KUKA KRL program: MyProgram_102().src

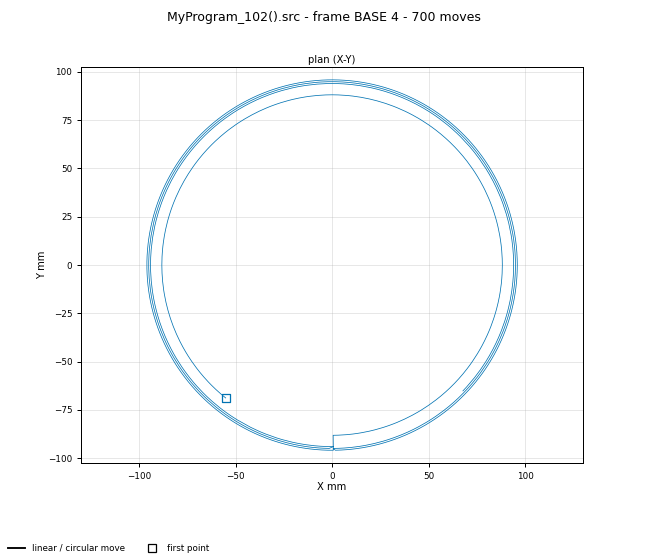
[picture p0: tool path of MyProgram_102().src in frame BASE 4, 700 of 700 moves have a stored position in this frame; points joined in program order, loops and branches not executed]
&ACCESS RVP
&REL 1
&PARAM TEMPLATE = C:\KRC\Roboter\Template\vorgabe
&PARAM EDITMASK = *
DEF MyProgram_102()
; ---- Setting reference (Base) ----
$BASE = BASE_DATA[4]

; --------------------------
; ---- Setting tool (TCP) ----
$TOOL = TOOL_DATA[3]
; --------------------------

$VEL.CP = VEL_APROX_PRINT
Startdeposition()
$VEL.CP = VEL_PRINT
LIN {X -55.0908,Y -68.8006,Z 92,A -133.8998,B 24.9282,C -1.9576,E1 24.8989,E2 -141.0227} C_DIS
LIN {X -57.6205,Y -66.6959,Z 92,A -136.0232,B 24.9278,C -1.9621,E1 24.8943,E2 -138.9019} C_DIS
LIN {X -60.1121,Y -64.4587,Z 92,A -138.1865,B 24.9275,C -1.9669,E1 24.8899,E2 -136.7412} C_DIS
LIN {X -62.4,Y -62.2469,Z 92,A -140.2884,B 24.9272,C -1.9702,E1 24.8857,E2 -134.6384} C_DIS
LIN {X -64.1532,Y -60.4369,Z 92,A -141.8968,B 24.9269,C -1.9746,E1 24.8826,E2 -133.0336} C_DIS
LIN {X -66.3939,Y -57.9664,Z 92,A -144.0684,B 24.9265,C -1.9794,E1 24.8786,E2 -130.8637} C_DIS
LIN {X -68.514,Y -55.4444,Z 92,A -146.1669,B 24.9261,C -1.9856,E1 24.8748,E2 -128.7703} C_DIS
LIN {X -70.1385,Y -53.3772,Z 92,A -147.8949,B 24.9258,C -1.9891,E1 24.8719,E2 -127.0425} C_DIS
LIN {X -71.5084,Y -51.5264,Z 92,A -149.3014,B 24.9253,C -1.9955,E1 24.8696,E2 -125.6443} C_DIS
LIN {X -72.6787,Y -49.8632,Z 92,A -150.8425,B 24.9256,C -1.9924,E1 24.8671,E2 -124.0882} C_DIS
LIN {X -74.4672,Y -47.1505,Z 92,A -152.7543,B 24.9247,C -2.0036,E1 24.8642,E2 -122.1936} C_DIS
LIN {X -75.8238,Y -44.9334,Z 92,A -154.6554,B 24.9249,C -2.002,E1 24.8615,E2 -120.2787} C_DIS
LIN {X -77.2426,Y -42.4507,Z 92,A -156.5523,B 24.9246,C -2.0058,E1 24.8589,E2 -118.3811} C_DIS
LIN {X -78.7875,Y -39.5087,Z 92,A -158.4218,B 24.9235,C -2.0202,E1 24.8565,E2 -116.5359} C_DIS
LIN {X -79.732,Y -37.5663,Z 92,A -159.8342,B 24.9232,C -2.0238,E1 24.8548,E2 -115.1246} C_DIS
LIN {X -80.5782,Y -35.7169,Z 92,A -161.3104,B 24.9232,C -2.0231,E1 24.8531,E2 -113.6385} C_DIS
LIN {X -81.475,Y -33.6191,Z 92,A -162.7506,B 24.9228,C -2.0286,E1 24.8516,E2 -112.2034} C_DIS
LIN {X -82.2377,Y -31.7093,Z 92,A -164.0784,B 24.9225,C -2.0327,E1 24.8502,E2 -110.878} C_DIS
LIN {X -83.0309,Y -29.5683,Z 92,A -165.5727,B 24.9222,C -2.0368,E1 24.8488,E2 -109.385} C_DIS
LIN {X -83.691,Y -27.6469,Z 92,A -166.9707,B 24.9221,C -2.0385,E1 24.8476,E2 -107.983} C_DIS
LIN {X -84.3756,Y -25.4792,Z 92,A -168.4079,B 24.9216,C -2.0441,E1 24.8464,E2 -106.5509} C_DIS
LIN {X -84.9491,Y -23.4984,Z 92,A -169.9139,B 24.9217,C -2.0434,E1 24.8452,E2 -105.0346} C_DIS
LIN {X -85.5268,Y -21.2978,Z 92,A -171.2261,B 24.921,C -2.0527,E1 24.8443,E2 -103.7368} C_DIS
LIN {X -85.9938,Y -19.3285,Z 92,A -172.5544,B 24.9207,C -2.0563,E1 24.8435,E2 -102.4095} C_DIS
LIN {X -86.4685,Y -17.077,Z 92,A -174.0675,B 24.9204,C -2.0605,E1 24.8427,E2 -100.8973} C_DIS
LIN {X -86.8426,Y -15.0633,Z 92,A -175.4002,B 24.9201,C -2.0646,E1 24.842,E2 -99.5665} C_DIS
LIN {X -87.1856,Y -12.931,Z 92,A -176.8138,B 24.9197,C -2.0687,E1 24.8414,E2 -98.1543} C_DIS
LIN {X -87.4909,Y -10.6657,Z 92,A -178.3106,B 24.9194,C -2.0731,E1 24.8409,E2 -96.659} C_DIS
LIN {X -87.726,Y -8.5188,Z 92,A -179.6515,B 24.9189,C -2.0793,E1 24.8405,E2 -95.3249} C_DIS
LIN {X -87.9265,Y -6.0991,Z 92,A 178.8138,B 24.9184,C -2.0855,E1 24.8401,E2 -93.7959} C_DIS
LIN {X -88.0388,Y -4.1929,Z 92,A 177.5128,B 24.9183,C -2.0878,E1 24.8399,E2 -92.4925} C_DIS
LIN {X -88.1151,Y -2.0351,Z 92,A 176.0233,B 24.9181,C -2.0898,E1 24.8399,E2 -90.9988} C_DIS
LIN {X -88.139,Y -0.0018,Z 92,A 174.7078,B 24.9178,C -2.0942,E1 24.8398,E2 -89.6858} C_DIS
LIN {X -88.1091,Y 2.2827,Z 92,A 173.2673,B 24.9173,C -2.1002,E1 24.8398,E2 -88.2511} C_DIS
LIN {X -88.0328,Y 4.3304,Z 92,A 171.7854,B 24.9173,C -2.1002,E1 24.84,E2 -86.7603} C_DIS
LIN {X -87.8451,Y 7.1771,Z 92,A 169.9225,B 24.9168,C -2.106,E1 24.8404,E2 -84.8999} C_DIS
LIN {X -87.6023,Y 9.7143,Z 92,A 168.2489,B 24.9164,C -2.1108,E1 24.8409,E2 -83.2277} C_DIS
LIN {X -87.3205,Y 11.9815,Z 92,A 166.5136,B 24.9166,C -2.1085,E1 24.8415,E2 -81.4766} C_DIS
LIN {X -86.8138,Y 15.2235,Z 92,A 164.4771,B 24.9159,C -2.118,E1 24.8425,E2 -79.4507} C_DIS
LIN {X -86.1961,Y 18.4018,Z 92,A 162.6299,B 24.9148,C -2.132,E1 24.8435,E2 -77.6259} C_DIS
LIN {X -85.7502,Y 20.3818,Z 92,A 161.158,B 24.9148,C -2.1318,E1 24.8444,E2 -76.1451} C_DIS
LIN {X -85.1932,Y 22.595,Z 92,A 159.8078,B 24.9141,C -2.1403,E1 24.8453,E2 -74.8072} C_DIS
LIN {X -84.6148,Y 24.6728,Z 92,A 158.2368,B 24.9141,C -2.1399,E1 24.8466,E2 -73.226} C_DIS
LIN {X -83.6925,Y 27.6422,Z 92,A 156.2829,B 24.9135,C -2.1481,E1 24.8482,E2 -71.2805} C_DIS
LIN {X -82.9482,Y 29.7998,Z 92,A 154.7907,B 24.9131,C -2.1524,E1 24.8496,E2 -69.7902} C_DIS
LIN {X -82.0355,Y 32.2245,Z 92,A 152.9841,B 24.913,C -2.1541,E1 24.8514,E2 -67.9775} C_DIS
LIN {X -80.8405,Y 35.1151,Z 92,A 151.1415,B 24.912,C -2.1657,E1 24.8534,E2 -66.1523} C_DIS
LIN {X -79.6031,Y 37.8382,Z 92,A 149.1721,B 24.9116,C -2.1708,E1 24.8557,E2 -64.1843} C_DIS
LIN {X -78.7225,Y 39.6396,Z 92,A 147.6445,B 24.9118,C -2.1682,E1 24.8576,E2 -62.6423} C_DIS
LIN {X -77.6641,Y 41.6736,Z 92,A 146.2785,B 24.9112,C -2.1761,E1 24.8593,E2 -61.2879} C_DIS
LIN {X -76.6219,Y 43.5602,Z 92,A 144.9444,B 24.9107,C -2.1821,E1 24.8612,E2 -59.9611} C_DIS
LIN {X -75.5337,Y 45.4211,Z 92,A 143.5333,B 24.9104,C -2.1858,E1 24.8632,E2 -58.5516} C_DIS
LIN {X -74.4003,Y 47.2548,Z 92,A 141.9678,B 24.9104,C -2.1851,E1 24.8655,E2 -56.9763} C_DIS
LIN {X -73.1491,Y 49.1685,Z 92,A 140.635,B 24.9097,C -2.1936,E1 24.8675,E2 -55.6572} C_DIS
LIN {X -72.0234,Y 50.8046,Z 92,A 139.1962,B 24.9098,C -2.1929,E1 24.8698,E2 -54.2096} C_DIS
LIN {X -70.701,Y 52.6286,Z 92,A 137.6109,B 24.9098,C -2.1934,E1 24.8725,E2 -52.6178} C_DIS
LIN {X -68.8213,Y 55.065,Z 92,A 135.5536,B 24.9095,C -2.197,E1 24.876,E2 -50.5594} C_DIS
LIN {X -66.7411,Y 57.5688,Z 92,A 133.442,B 24.909,C -2.2026,E1 24.8798,E2 -48.4515} C_DIS
LIN {X -64.6768,Y 59.8775,Z 92,A 131.3966,B 24.9087,C -2.2067,E1 24.8837,E2 -46.4068} C_DIS
LIN {X -62.3288,Y 62.3189,Z 92,A 129.1613,B 24.9083,C -2.211,E1 24.888,E2 -44.1723} C_DIS
LIN {X -60.3328,Y 64.2511,Z 92,A 127.3713,B 24.9079,C -2.2157,E1 24.8917,E2 -42.3862} C_DIS
LIN {X -57.8348,Y 66.5088,Z 92,A 125.2447,B 24.9073,C -2.2225,E1 24.8961,E2 -40.2673} C_DIS
LIN {X -55.4085,Y 68.5431,Z 92,A 123.1721,B 24.907,C -2.2266,E1 24.9005,E2 -38.1966} C_DIS
LIN {X -53.2048,Y 70.2681,Z 92,A 121.5765,B 24.9061,C -2.237,E1 24.904,E2 -36.6199} C_DIS
LIN {X -51.4953,Y 71.5306,Z 92,A 120.1031,B 24.9061,C -2.2371,E1 24.9074,E2 -35.1416} C_DIS
LIN {X -49.8396,Y 72.6947,Z 92,A 118.7813,B 24.9059,C -2.2395,E1 24.9104,E2 -33.8211} C_DIS
LIN {X -48.05,Y 73.8899,Z 92,A 117.1497,B 24.9063,C -2.2354,E1 24.9142,E2 -32.1742} C_DIS
LIN {X -45.2023,Y 75.6648,Z 92,A 115.2604,B 24.9052,C -2.248,E1 24.9187,E2 -30.3092} C_DIS
LIN {X -43.4499,Y 76.6853,Z 92,A 113.8593,B 24.9052,C -2.2479,E1 24.9221,E2 -28.9035} C_DIS
LIN {X -41.4529,Y 77.7823,Z 92,A 112.3756,B 24.905,C -2.2503,E1 24.9257,E2 -27.4215} C_DIS
LIN {X -39.508,Y 78.7879,Z 92,A 111.0212,B 24.9046,C -2.2547,E1 24.9291,E2 -26.0738} C_DIS
LIN {X -37.5665,Y 79.7319,Z 92,A 109.6134,B 24.9045,C -2.2567,E1 24.9326,E2 -24.6673} C_DIS
LIN {X -35.7178,Y 80.5778,Z 92,A 108.0849,B 24.9048,C -2.2525,E1 24.9365,E2 -23.125} C_DIS
LIN {X -33.7201,Y 81.4339,Z 92,A 106.7186,B 24.9045,C -2.2559,E1 24.94,E2 -21.7637} C_DIS
LIN {X -31.6873,Y 82.2461,Z 92,A 105.3688,B 24.9042,C -2.26,E1 24.9435,E2 -20.4208} C_DIS
LIN {X -29.2147,Y 83.155,Z 92,A 103.5195,B 24.9043,C -2.2581,E1 24.9484,E2 -18.5632} C_DIS
LIN {X -26.4901,Y 84.0636,Z 92,A 101.8544,B 24.9036,C -2.2664,E1 24.9528,E2 -16.9148} C_DIS
LIN {X -24.4281,Y 84.6858,Z 92,A 100.4479,B 24.9036,C -2.2677,E1 24.9566,E2 -15.5091} C_DIS
LIN {X -22.4732,Y 85.2261,Z 92,A 98.9898,B 24.9038,C -2.2648,E1 24.9605,E2 -14.0418} C_DIS
LIN {X -20.2625,Y 85.778,Z 92,A 97.4007,B 24.9039,C -2.2629,E1 24.9648,E2 -12.4461} C_DIS
LIN {X -17.1934,Y 86.4461,Z 92,A 95.2808,B 24.9039,C -2.2622,E1 24.9706,E2 -10.3221} C_DIS
LIN {X -13.9877,Y 87.0222,Z 92,A 93.4019,B 24.9032,C -2.2711,E1 24.9758,E2 -8.4624} C_DIS
LIN {X -11.8524,Y 87.3387,Z 92,A 91.9278,B 24.9033,C -2.2698,E1 24.9799,E2 -6.984} C_DIS
LIN {X -9.5843,Y 87.6159,Z 92,A 90.5083,B 24.9031,C -2.2727,E1 24.9838,E2 -5.5705} C_DIS
LIN {X -7.561,Y 87.8144,Z 92,A 89.0193,B 24.9035,C -2.2681,E1 24.9879,E2 -4.0699} C_DIS
LIN {X -5.258,Y 87.9816,Z 92,A 87.6833,B 24.903,C -2.2739,E1 24.9916,E2 -2.7471} C_DIS
LIN {X -3.2295,Y 88.08,Z 92,A 86.1609,B 24.9035,C -2.268,E1 24.9959,E2 -1.2104} C_DIS
LIN {X 0.0063,Y 88.1393,Z 92,A 84.0319,B 24.9035,C -2.2677,E1 25.0019,E2 0.9194} C_DIS
LIN {X 3.2426,Y 88.0796,Z 92,A 82.1507,B 24.9029,C -2.2749,E1 25.0071,E2 2.783} C_DIS
LIN {X 5.712,Y 87.9527,Z 92,A 80.6353,B 24.9027,C -2.2778,E1 25.0113,E2 4.2909} C_DIS
LIN {X 7.6239,Y 87.8086,Z 92,A 79.1484,B 24.9033,C -2.2701,E1 25.0155,E2 5.7953} C_DIS
LIN {X 10.6692,Y 87.4905,Z 92,A 77.2297,B 24.9031,C -2.2721,E1 25.0208,E2 7.708} C_DIS
LIN {X 13.059,Y 87.1658,Z 92,A 75.741,B 24.903,C -2.2742,E1 25.0249,E2 9.1903} C_DIS
LIN {X 15.0667,Y 86.842,Z 92,A 74.4194,B 24.903,C -2.2738,E1 25.0285,E2 10.5117} C_DIS
LIN {X 17.3273,Y 86.4186,Z 92,A 72.811,B 24.9034,C -2.2695,E1 25.0329,E2 12.1282} C_DIS
LIN {X 19.4335,Y 85.9695,Z 92,A 71.5506,B 24.903,C -2.2733,E1 25.0363,E2 13.378} C_DIS
LIN {X 21.5838,Y 85.4548,Z 92,A 70.1059,B 24.9031,C -2.2722,E1 25.0403,E2 14.8231} C_DIS
LIN {X 23.5283,Y 84.9408,Z 92,A 68.7213,B 24.9034,C -2.2689,E1 25.044,E2 16.2135} C_DIS
LIN {X 25.5972,Y 84.3404,Z 92,A 67.3223,B 24.9035,C -2.2679,E1 25.0478,E2 17.6123} C_DIS
LIN {X 27.6515,Y 83.6895,Z 92,A 65.9918,B 24.9035,C -2.2691,E1 25.0513,E2 18.9376} C_DIS
LIN {X 29.8076,Y 82.9453,Z 92,A 64.4996,B 24.9035,C -2.2675,E1 25.0552,E2 20.4305} C_DIS
LIN {X 31.7317,Y 82.2291,Z 92,A 63.1111,B 24.9038,C -2.2644,E1 25.0588,E2 21.8233} C_DIS
LIN {X 33.7362,Y 81.4273,Z 92,A 61.7105,B 24.9039,C -2.2631,E1 25.0625,E2 23.2238} C_DIS
LIN {X 35.8356,Y 80.5247,Z 92,A 60.3722,B 24.9036,C -2.2663,E1 25.0659,E2 24.5513} C_DIS
LIN {X 37.7974,Y 79.6227,Z 92,A 58.9707,B 24.9038,C -2.2647,E1 25.0694,E2 25.953} C_DIS
LIN {X 39.6242,Y 78.7303,Z 92,A 57.5772,B 24.9041,C -2.2607,E1 25.0729,E2 27.3523} C_DIS
LIN {X 41.6636,Y 77.6695,Z 92,A 55.9506,B 24.9047,C -2.2544,E1 25.077,E2 28.9892} C_DIS
LIN {X 44.3912,Y 76.1443,Z 92,A 53.9967,B 24.9047,C -2.2541,E1 25.0817,E2 30.938} C_DIS
LIN {X 46.2391,Y 75.0365,Z 92,A 52.4841,B 24.9052,C -2.2482,E1 25.0853,E2 32.4596} C_DIS
LIN {X 48.1741,Y 73.8084,Z 92,A 51.1819,B 24.9048,C -2.2521,E1 25.0883,E2 33.7484} C_DIS
LIN {X 49.969,Y 72.6052,Z 92,A 49.7984,B 24.905,C -2.2506,E1 25.0915,E2 35.1309} C_DIS
LIN {X 51.792,Y 71.3158,Z 92,A 48.3444,B 24.9052,C -2.248,E1 25.0948,E2 36.586} C_DIS
LIN {X 53.8698,Y 69.7589,Z 92,A 46.5669,B 24.9057,C -2.242,E1 25.0988,E2 38.3711} C_DIS
LIN {X 56.3278,Y 67.7896,Z 92,A 44.4846,B 24.9061,C -2.237,E1 25.1033,E2 40.4574} C_DIS
LIN {X 58.7884,Y 65.6672,Z 92,A 42.4033,B 24.9064,C -2.2339,E1 25.1077,E2 42.5378} C_DIS
LIN {X 61.1617,Y 63.4625,Z 92,A 40.3127,B 24.9067,C -2.2301,E1 25.1119,E2 44.6288} C_DIS
LIN {X 63.584,Y 61.0357,Z 92,A 38.0714,B 24.9071,C -2.2249,E1 25.1163,E2 46.8728} C_DIS
LIN {X 65.6906,Y 58.7622,Z 92,A 36.0882,B 24.9074,C -2.2215,E1 25.1201,E2 48.8552} C_DIS
LIN {X 67.7931,Y 56.3236,Z 92,A 33.9988,B 24.9078,C -2.2168,E1 25.1238,E2 50.9463} C_DIS
LIN {X 69.8171,Y 53.7943,Z 92,A 31.9054,B 24.9082,C -2.2122,E1 25.1275,E2 53.0407} C_DIS
LIN {X 71.5065,Y 51.5289,Z 92,A 30.1759,B 24.9082,C -2.2114,E1 25.1303,E2 54.7639} C_DIS
LIN {X 72.6868,Y 49.8513,Z 92,A 28.8639,B 24.9085,C -2.2087,E1 25.1324,E2 56.0757} C_DIS
LIN {X 73.8818,Y 48.0627,Z 92,A 27.4051,B 24.909,C -2.2031,E1 25.1346,E2 57.5406} C_DIS
LIN {X 75.336,Y 45.7465,Z 92,A 25.6046,B 24.9094,C -2.1977,E1 25.1373,E2 59.3447} C_DIS
LIN {X 76.8415,Y 43.1704,Z 92,A 23.6162,B 24.91,C -2.1908,E1 25.1401,E2 61.3391} C_DIS
LIN {X 78.2963,Y 40.4734,Z 92,A 21.7949,B 24.91,C -2.1912,E1 25.1424,E2 63.1497} C_DIS
LIN {X 79.2093,Y 38.6577,Z 92,A 20.4139,B 24.9104,C -2.1855,E1 25.1442,E2 64.537} C_DIS
LIN {X 80.2289,Y 36.4919,Z 92,A 19.0306,B 24.9103,C -2.1871,E1 25.1458,E2 65.9089} C_DIS
LIN {X 81.0773,Y 34.5667,Z 92,A 17.6529,B 24.9106,C -2.1828,E1 25.1473,E2 67.2891} C_DIS
LIN {X 81.894,Y 32.5847,Z 92,A 16.2686,B 24.9109,C -2.1791,E1 25.1488,E2 68.6745} C_DIS
LIN {X 82.8407,Y 30.0945,Z 92,A 14.2939,B 24.912,C -2.1656,E1 25.1507,E2 70.6702} C_DIS
LIN {X 83.6873,Y 27.6579,Z 92,A 12.5817,B 24.9125,C -2.1594,E1 25.1522,E2 72.3875} C_DIS
LIN {X 84.6867,Y 24.4251,Z 92,A 10.6947,B 24.9122,C -2.1637,E1 25.1537,E2 74.2535} C_DIS
LIN {X 85.2283,Y 22.465,Z 92,A 9.2385,B 24.9129,C -2.1549,E1 25.1548,E2 75.7219} C_DIS
LIN {X 85.8933,Y 19.7634,Z 92,A 7.4194,B 24.9134,C -2.1491,E1 25.156,E2 77.5444} C_DIS
LIN {X 86.4709,Y 17.0642,Z 92,A 5.7273,B 24.9135,C -2.1471,E1 25.1569,E2 79.2314} C_DIS
LIN {X 86.8421,Y 15.0658,Z 92,A 4.4151,B 24.9138,C -2.1433,E1 25.1576,E2 80.5449} C_DIS
LIN {X 87.1851,Y 12.9345,Z 92,A 3.0201,B 24.9142,C -2.1391,E1 25.1582,E2 81.9414} C_DIS
LIN {X 87.5401,Y 10.2459,Z 92,A 1.1621,B 24.9149,C -2.1303,E1 25.1588,E2 83.8093} C_DIS
LIN {X 87.8161,Y 7.5401,Z 92,A -0.4838,B 24.9149,C -2.1289,E1 25.1593,E2 85.4486} C_DIS
LIN {X 87.9811,Y 5.2664,Z 92,A -1.9741,B 24.9154,C -2.1239,E1 25.1596,E2 86.9419} C_DIS
LIN {X 88.0797,Y 3.24,Z 92,A -3.4659,B 24.9162,C -2.1136,E1 25.1597,E2 88.4491} C_DIS
LIN {X 88.1389,Y 0.0069,Z 92,A -5.3507,B 24.9162,C -2.1145,E1 25.1597,E2 90.3205} C_DIS
LIN {X 88.1084,Y -2.3048,Z 92,A -6.7714,B 24.9162,C -2.1126,E1 25.1597,E2 91.7373} C_DIS
LIN {X 88.0326,Y -4.3342,Z 92,A -8.2242,B 24.917,C -2.1037,E1 25.1595,E2 93.2026} C_DIS
LIN {X 87.8575,Y -7.0222,Z 92,A -10.0056,B 24.9175,C -2.097,E1 25.1592,E2 94.9892} C_DIS
LIN {X 87.6028,Y -9.7095,Z 92,A -11.7033,B 24.9178,C -2.0934,E1 25.1587,E2 96.6854} C_DIS
LIN {X 87.29,Y -12.1961,Z 92,A -13.154,B 24.9178,C -2.0945,E1 25.1582,E2 98.125} C_DIS
LIN {X 86.9984,Y -14.1314,Z 92,A -14.4445,B 24.9181,C -2.0897,E1 25.1576,E2 99.4191} C_DIS
LIN {X 86.5651,Y -16.575,Z 92,A -16.2682,B 24.9191,C -2.0772,E1 25.1567,E2 101.2617} C_DIS
LIN {X 85.912,Y -19.6825,Z 92,A -18.3634,B 24.9197,C -2.0695,E1 25.1554,E2 103.3627} C_DIS
LIN {X 85.1708,Y -22.6778,Z 92,A -20.0757,B 24.9194,C -2.0735,E1 25.1543,E2 105.0557} C_DIS
LIN {X 84.5682,Y -24.8298,Z 92,A -21.7542,B 24.9203,C -2.061,E1 25.153,E2 106.7541} C_DIS
LIN {X 83.6823,Y -27.6728,Z 92,A -23.5261,B 24.9203,C -2.0607,E1 25.1515,E2 108.5167} C_DIS
LIN {X 82.9399,Y -29.8225,Z 92,A -24.9955,B 24.9207,C -2.0565,E1 25.1501,E2 109.9879} C_DIS
LIN {X 82.2338,Y -31.7197,Z 92,A -26.3809,B 24.9212,C -2.05,E1 25.1487,E2 111.381} C_DIS
LIN {X 81.4257,Y -33.7399,Z 92,A -27.7764,B 24.9215,C -2.0463,E1 25.1472,E2 112.7774} C_DIS
LIN {X 80.3531,Y -36.2164,Z 92,A -29.5599,B 24.922,C -2.04,E1 25.1452,E2 114.566} C_DIS
LIN {X 78.959,Y -39.1628,Z 92,A -31.6587,B 24.9224,C -2.0344,E1 25.1427,E2 116.6667} C_DIS
LIN {X 77.6798,Y -41.6448,Z 92,A -33.3604,B 24.9224,C -2.033,E1 25.1405,E2 118.3628} C_DIS
LIN {X 76.6385,Y -43.5313,Z 92,A -34.6938,B 24.9226,C -2.0313,E1 25.1387,E2 119.6933} C_DIS
LIN {X 75.271,Y -45.8533,Z 92,A -36.6436,B 24.9235,C -2.0194,E1 25.1358,E2 121.6612} C_DIS
LIN {X 73.8066,Y -48.1767,Z 92,A -38.2687,B 24.9235,C -2.0199,E1 25.1334,E2 123.2769} C_DIS
LIN {X 72.6762,Y -49.8669,Z 92,A -39.5825,B 24.9238,C -2.0165,E1 25.1313,E2 124.5923} C_DIS
LIN {X 71.3581,Y -51.7343,Z 92,A -41.0595,B 24.924,C -2.0127,E1 25.1289,E2 126.0709} C_DIS
LIN {X 69.7778,Y -53.8452,Z 92,A -42.8608,B 24.9246,C -2.0051,E1 25.1259,E2 127.8817} C_DIS
LIN {X 67.7817,Y -56.3373,Z 92,A -44.9696,B 24.9251,C -1.9985,E1 25.1222,E2 129.9963} C_DIS
LIN {X 65.666,Y -58.7897,Z 92,A -47.0296,B 24.9254,C -1.9947,E1 25.1184,E2 132.0561} C_DIS
LIN {X 63.4614,Y -61.1628,Z 92,A -49.1654,B 24.9259,C -1.9884,E1 25.1143,E2 134.1974} C_DIS
LIN {X 61.1128,Y -63.5097,Z 92,A -51.2854,B 24.9262,C -1.9845,E1 25.11,E2 136.3177} C_DIS
LIN {X 58.7852,Y -65.67,Z 92,A -53.3251,B 24.9265,C -1.9806,E1 25.1058,E2 138.3585} C_DIS
LIN {X 56.3325,Y -67.7856,Z 92,A -55.4211,B 24.9268,C -1.9762,E1 25.1014,E2 140.4568} C_DIS
LIN {X 53.7912,Y -69.8194,Z 92,A -57.5281,B 24.9271,C -1.9719,E1 25.0967,E2 142.5661} C_DIS
LIN {X 51.4464,Y -71.5654,Z 92,A -59.259,B 24.927,C -1.9737,E1 25.0929,E2 144.2865} C_DIS
LIN {X 49.8621,Y -72.6795,Z 92,A -60.5632,B 24.9273,C -1.9696,E1 25.0899,E2 145.5959} C_DIS
LIN {X 48.0665,Y -73.8793,Z 92,A -62.0278,B 24.9276,C -1.9648,E1 25.0864,E2 147.067} C_DIS
LIN {X 46.242,Y -75.0347,Z 92,A -63.4242,B 24.9278,C -1.9624,E1 25.0831,E2 148.4646} C_DIS
LIN {X 44.3899,Y -76.145,Z 92,A -64.9802,B 24.9284,C -1.9547,E1 25.0793,E2 150.0341} C_DIS
LIN {X 41.4107,Y -77.8045,Z 92,A -66.9641,B 24.9281,C -1.9587,E1 25.0745,E2 152.0028} C_DIS
LIN {X 39.4966,Y -78.7935,Z 92,A -68.2853,B 24.9281,C -1.9591,E1 25.0712,E2 153.3195} C_DIS
LIN {X 37.5579,Y -79.7359,Z 92,A -69.6812,B 24.9281,C -1.957,E1 25.0677,E2 154.7167} C_DIS
LIN {X 35.7116,Y -80.5805,Z 92,A -71.1398,B 24.9287,C -1.9503,E1 25.064,E2 156.1874} C_DIS
LIN {X 33.7294,Y -81.4301,Z 92,A -72.5532,B 24.9289,C -1.9479,E1 25.0603,E2 157.6033} C_DIS
LIN {X 31.6997,Y -82.2414,Z 92,A -73.8839,B 24.9288,C -1.949,E1 25.0569,E2 158.9286} C_DIS
LIN {X 29.0976,Y -83.196,Z 92,A -75.8259,B 24.9293,C -1.942,E1 25.0518,E2 160.8831} C_DIS
LIN {X 26.4171,Y -84.0862,Z 92,A -77.4318,B 24.9289,C -1.9474,E1 25.0475,E2 162.4732} C_DIS
LIN {X 24.3899,Y -84.6966,Z 92,A -78.9383,B 24.9293,C -1.9415,E1 25.0435,E2 163.9909} C_DIS
LIN {X 22.1945,Y -85.2978,Z 92,A -80.5261,B 24.9297,C -1.9364,E1 25.0392,E2 165.5884} C_DIS
LIN {X 19.3017,Y -85.9998,Z 92,A -82.295,B 24.9294,C -1.94,E1 25.0344,E2 167.3462} C_DIS
LIN {X 17.0652,Y -86.4708,Z 92,A -83.7782,B 24.9295,C -1.9388,E1 25.0303,E2 168.8304} C_DIS
LIN {X 15.066,Y -86.8421,Z 92,A -85.0977,B 24.9295,C -1.9378,E1 25.0267,E2 170.1508} C_DIS
LIN {X 12.9099,Y -87.1886,Z 92,A -86.514,B 24.9297,C -1.9369,E1 25.0228,E2 171.5679} C_DIS
LIN {X 10.6476,Y -87.4931,Z 92,A -88.1087,B 24.93,C -1.9324,E1 25.0183,E2 173.1722} C_DIS
LIN {X 7.554,Y -87.815,Z 92,A -90.0157,B 24.9298,C -1.935,E1 25.0131,E2 175.0718} C_DIS
LIN {X 5.2762,Y -87.9806,Z 92,A -91.4994,B 24.9298,C -1.9344,E1 25.0089,E2 176.5562} C_DIS
LIN {X 3.2145,Y -88.0805,Z 92,A -92.9054,B 24.93,C -1.9318,E1 25.005,E2 177.9679} C_DIS
LIN {X 0.5522,Y -88.1352,Z 92,A -94.3295,B 24.9293,C -1.9413,E1 25.0011,E2 179.3694} C_DIS
Enddeposition()
LIN {X 0.6522,Y -95.88,Z 93,A -93.6861,B 24.937,C -1.8339,E1 25.0022,E2 178.9806} C_DIS
Startdeposition()
$VEL.CP = VEL_PRINT
LIN {X -2.3531,Y -95.8559,Z 93,A -96.0515,B 24.9384,C -1.8132,E1 24.9954,E2 181.3953} C_DIS
LIN {X -5.2153,Y -95.7411,Z 93,A -97.8055,B 24.9384,C -1.8116,E1 24.9905,E2 183.1535} C_DIS
LIN {X -8.2267,Y -95.5312,Z 93,A -99.5668,B 24.9384,C -1.8131,E1 24.9856,E2 184.912} C_DIS
LIN {X -11.0764,Y -95.2411,Z 93,A -101.3215,B 24.9384,C -1.8118,E1 24.9807,E2 186.6707} C_DIS
LIN {X -13.5631,Y -94.9189,Z 93,A -102.7783,B 24.9384,C -1.8136,E1 24.9767,E2 188.1246} C_DIS
LIN {X -16.3926,Y -94.4731,Z 93,A -104.4911,B 24.9384,C -1.814,E1 24.972,E2 189.8379} C_DIS
LIN {X -19.2069,Y -93.9396,Z 93,A -106.2468,B 24.9384,C -1.8131,E1 24.9672,E2 191.5975} C_DIS
LIN {X -22.155,Y -93.2901,Z 93,A -108.0098,B 24.9382,C -1.8154,E1 24.9624,E2 193.3574} C_DIS
LIN {X -24.4377,Y -92.7183,Z 93,A -109.4179,B 24.9382,C -1.8162,E1 24.9586,E2 194.7658} C_DIS
LIN {X -26.7058,Y -92.0907,Z 93,A -110.996,B 24.9385,C -1.8112,E1 24.9543,E2 196.3583} C_DIS
LIN {X -29.5909,Y -91.2027,Z 93,A -112.6331,B 24.938,C -1.8183,E1 24.95,E2 197.9814} C_DIS
LIN {X -31.8203,Y -90.449,Z 93,A -114.0418,B 24.938,C -1.8193,E1 24.9462,E2 199.3903} C_DIS
LIN {X -34.0304,Y -89.6409,Z 93,A -115.5364,B 24.938,C -1.8176,E1 24.9423,E2 200.8921} C_DIS
LIN {X -37.1646,Y -88.3875,Z 93,A -117.5151,B 24.9378,C -1.8209,E1 24.9372,E2 202.8673} C_DIS
LIN {X -39.9293,Y -87.1754,Z 93,A -119.3547,B 24.9378,C -1.8217,E1 24.9325,E2 204.7096} C_DIS
LIN {X -42.6529,Y -85.8737,Z 93,A -121.0894,B 24.9375,C -1.8262,E1 24.9282,E2 206.438} C_DIS
LIN {X -44.7475,Y -84.801,Z 93,A -122.5852,B 24.9375,C -1.825,E1 24.9244,E2 207.9409} C_DIS
LIN {X -47.7047,Y -83.1734,Z 93,A -124.5655,B 24.9373,C -1.829,E1 24.9196,E2 209.9174} C_DIS
LIN {X -50.3002,Y -81.632,Z 93,A -126.5296,B 24.9375,C -1.8262,E1 24.9149,E2 211.8941} C_DIS
LIN {X -52.844,Y -80.0067,Z 93,A -128.1425,B 24.9369,C -1.8354,E1 24.9112,E2 213.4903} C_DIS
LIN {X -55.2112,Y -78.3939,Z 93,A -129.8601,B 24.9367,C -1.838,E1 24.9072,E2 215.2076} C_DIS
LIN {X -57.3769,Y -76.8213,Z 93,A -131.5722,B 24.9367,C -1.837,E1 24.9033,E2 216.928} C_DIS
LIN {X -59.5135,Y -75.1778,Z 93,A -133.083,B 24.9363,C -1.8432,E1 24.9,E2 218.4296} C_DIS
LIN {X -61.7337,Y -73.3679,Z 93,A -134.9991,B 24.9366,C -1.8397,E1 24.8959,E2 220.3615} C_DIS
LIN {X -64.0114,Y -71.3869,Z 93,A -136.699,B 24.9361,C -1.8466,E1 24.8924,E2 222.0516} C_DIS
LIN {X -66.1164,Y -69.4443,Z 93,A -138.5301,B 24.9361,C -1.8462,E1 24.8886,E2 223.8913} C_DIS
LIN {X -68.2685,Y -67.3273,Z 93,A -140.1448,B 24.9354,C -1.8562,E1 24.8855,E2 225.4889} C_DIS
LIN {X -70.2504,Y -65.2593,Z 93,A -142.0624,B 24.9356,C -1.8532,E1 24.8817,E2 227.4222} C_DIS
LIN {X -72.2685,Y -63.0144,Z 93,A -143.7635,B 24.9351,C -1.8606,E1 24.8786,E2 229.1131} C_DIS
LIN {X -74.5009,Y -60.3586,Z 93,A -145.8651,B 24.9348,C -1.8645,E1 24.8749,E2 231.2152} C_DIS
LIN {X -76.3087,Y -58.0593,Z 93,A -147.7163,B 24.9348,C -1.8653,E1 24.8717,E2 233.0732} C_DIS
LIN {X -78.097,Y -55.6274,Z 93,A -149.4182,B 24.9342,C -1.8731,E1 24.8689,E2 234.7648} C_DIS
LIN {X -80.0067,Y -52.844,Z 93,A -151.4035,B 24.9338,C -1.8793,E1 24.8658,E2 236.7453} C_DIS
LIN {X -81.3612,Y -50.7337,Z 93,A -152.8676,B 24.9334,C -1.8842,E1 24.8637,E2 238.205} C_DIS
LIN {X -82.6496,Y -48.6069,Z 93,A -154.5508,B 24.9336,C -1.8818,E1 24.8612,E2 239.9027} C_DIS
LIN {X -84.3191,Y -45.6491,Z 93,A -156.49,B 24.933,C -1.8902,E1 24.8586,E2 241.832} C_DIS
LIN {X -85.6466,Y -43.1109,Z 93,A -158.3238,B 24.933,C -1.891,E1 24.8563,E2 243.6738} C_DIS
LIN {X -86.9597,Y -40.3927,Z 93,A -159.9869,B 24.9323,C -1.9006,E1 24.8543,E2 245.3231} C_DIS
LIN {X -88.129,Y -37.7778,Z 93,A -161.8614,B 24.9323,C -1.9002,E1 24.8522,E2 247.2088} C_DIS
LIN {X -89.2729,Y -34.9843,Z 93,A -163.5397,B 24.9316,C -1.9095,E1 24.8505,E2 248.8744} C_DIS
LIN {X -90.2798,Y -32.3026,Z 93,A -165.2018,B 24.9312,C -1.916,E1 24.8489,E2 250.5302} C_DIS
LIN {X -91.2027,Y -29.5909,Z 93,A -166.9675,B 24.9309,C -1.9194,E1 24.8473,E2 252.2979} C_DIS
LIN {X -91.9453,Y -27.1959,Z 93,A -168.4331,B 24.9305,C -1.925,E1 24.8461,E2 253.7586} C_DIS
LIN {X -92.585,Y -24.9312,Z 93,A -169.8486,B 24.9302,C -1.929,E1 24.8451,E2 255.1729} C_DIS
LIN {X -93.2901,Y -22.155,Z 93,A -171.7701,B 24.9303,C -1.9275,E1 24.8438,E2 257.1091} C_DIS
LIN {X -93.9396,Y -19.2069,Z 93,A -173.3883,B 24.9295,C -1.939,E1 24.8429,E2 258.7095} C_DIS
LIN {X -94.4731,Y -16.3926,Z 93,A -175.112,B 24.9292,C -1.9439,E1 24.842,E2 260.4316} C_DIS
LIN {X -94.9258,Y -13.5143,Z 93,A -176.9825,B 24.9291,C -1.9453,E1 24.8412,E2 262.3099} C_DIS
LIN {X -95.3158,Y -10.4234,Z 93,A -178.915,B 24.9288,C -1.949,E1 24.8406,E2 264.2453} C_DIS
LIN {X -95.5843,Y -7.5633,Z 93,A 179.4457,B 24.9282,C -1.9569,E1 24.8402,E2 265.8756} C_DIS
LIN {X -95.7693,Y -4.7048,Z 93,A 177.6898,B 24.9279,C -1.9609,E1 24.8399,E2 267.6325} C_DIS
LIN {X -95.8682,Y -1.6878,Z 93,A 175.9675,B 24.9273,C -1.9693,E1 24.8398,E2 269.3451} C_DIS
LIN {X -95.8682,Y 1.6878,Z 93,A 173.917,B 24.9269,C -1.9747,E1 24.8398,E2 271.395} C_DIS
LIN {X -95.7693,Y 4.7048,Z 93,A 171.9453,B 24.9269,C -1.9752,E1 24.8401,E2 273.3775} C_DIS
LIN {X -95.572,Y 7.7171,Z 93,A 170.2404,B 24.9262,C -1.9841,E1 24.8404,E2 275.0713} C_DIS
LIN {X -95.2411,Y 11.0764,Z 93,A 168.2523,B 24.9256,C -1.9915,E1 24.841,E2 277.0537} C_DIS
LIN {X -94.9189,Y 13.5631,Z 93,A 166.7858,B 24.9252,C -1.9973,E1 24.8415,E2 278.5151} C_DIS
LIN {X -94.4731,Y 16.3926,Z 93,A 165.0622,B 24.9248,C -2.0024,E1 24.8423,E2 280.2369} C_DIS
LIN {X -93.9396,Y 19.2069,Z 93,A 163.2955,B 24.9245,C -2.0061,E1 24.8433,E2 282.0051} C_DIS
LIN {X -93.405,Y 21.6576,Z 93,A 161.7434,B 24.9243,C -2.0092,E1 24.8442,E2 283.5589} C_DIS
LIN {X -92.7183,Y 24.4377,Z 93,A 160.1059,B 24.9237,C -2.0169,E1 24.8453,E2 285.1876} C_DIS
LIN {X -92.0907,Y 26.7058,Z 93,A 158.6899,B 24.9234,C -2.021,E1 24.8464,E2 286.602} C_DIS
LIN {X -91.4076,Y 28.9578,Z 93,A 157.0758,B 24.9236,C -2.0188,E1 24.8478,E2 288.2306} C_DIS
LIN {X -90.449,Y 31.8203,Z 93,A 155.4577,B 24.9227,C -2.0303,E1 24.8492,E2 289.8305} C_DIS
LIN {X -89.6409,Y 34.0304,Z 93,A 154.0417,B 24.9224,C -2.0343,E1 24.8506,E2 291.2449} C_DIS
LIN {X -88.7787,Y 36.22,Z 93,A 152.5401,B 24.9224,C -2.0356,E1 24.8522,E2 292.7519} C_DIS
LIN {X -87.6588,Y 38.8565,Z 93,A 150.7051,B 24.9222,C -2.0368,E1 24.8542,E2 294.594} C_DIS
LIN {X -86.3906,Y 41.5959,Z 93,A 149.0011,B 24.9215,C -2.0454,E1 24.8562,E2 296.2869} C_DIS
LIN {X -85.1111,Y 44.1587,Z 93,A 147.1665,B 24.9215,C -2.0465,E1 24.8586,E2 298.1286} C_DIS
LIN {X -83.6773,Y 46.8151,Z 93,A 145.549,B 24.9206,C -2.0577,E1 24.8607,E2 299.7279} C_DIS
LIN {X -82.2431,Y 49.2946,Z 93,A 143.6284,B 24.9207,C -2.056,E1 24.8635,E2 301.6626} C_DIS
LIN {X -80.6491,Y 51.8582,Z 93,A 141.9252,B 24.9201,C -2.0643,E1 24.866,E2 303.3547} C_DIS
LIN {X -78.9618,Y 54.3943,Z 93,A 140.0188,B 24.9199,C -2.0665,E1 24.869,E2 305.2652} C_DIS
LIN {X -77.3174,Y 56.706,Z 93,A 138.3884,B 24.9194,C -2.0732,E1 24.8716,E2 306.8876} C_DIS
LIN {X -75.2735,Y 59.3924,Z 93,A 136.4025,B 24.9189,C -2.0796,E1 24.875,E2 308.8677} C_DIS
LIN {X -73.6946,Y 61.3405,Z 93,A 134.8524,B 24.9187,C -2.0818,E1 24.8778,E2 310.4196} C_DIS
LIN {X -71.8308,Y 63.5156,Z 93,A 133.0191,B 24.9187,C -2.0823,E1 24.8812,E2 312.2601} C_DIS
LIN {X -69.7945,Y 65.7441,Z 93,A 131.3171,B 24.9181,C -2.09,E1 24.8844,E2 313.9511} C_DIS
LIN {X -67.6439,Y 67.9557,Z 93,A 129.4042,B 24.9179,C -2.0922,E1 24.8881,E2 315.8669} C_DIS
LIN {X -65.6317,Y 69.9002,Z 93,A 127.7832,B 24.9175,C -2.0978,E1 24.8914,E2 317.4813} C_DIS
LIN {X -63.5582,Y 71.7927,Z 93,A 126.1815,B 24.917,C -2.1041,E1 24.8947,E2 319.0744} C_DIS
LIN {X -61.2915,Y 73.7353,Z 93,A 124.2773,B 24.917,C -2.1041,E1 24.8988,E2 320.9857} C_DIS
LIN {X -58.9914,Y 75.5904,Z 93,A 122.616,B 24.9164,C -2.1113,E1 24.9024,E2 322.6362} C_DIS
LIN {X -56.706,Y 77.3174,Z 93,A 120.8537,B 24.9162,C -2.1133,E1 24.9063,E2 324.4002} C_DIS
LIN {X -54.6648,Y 78.7738,Z 93,A 119.3057,B 24.9162,C -2.1147,E1 24.9099,E2 325.9502} C_DIS
LIN {X -52.2884,Y 80.373,Z 93,A 117.4749,B 24.9162,C -2.1141,E1 24.9142,E2 327.7885} C_DIS
LIN {X -49.7315,Y 81.9776,Z 93,A 115.8609,B 24.9154,C -2.1236,E1 24.9179,E2 329.3847} C_DIS
LIN {X -47.2614,Y 83.4281,Z 93,A 114.1427,B 24.9152,C -2.1264,E1 24.9221,E2 331.1014} C_DIS
LIN {X -45.1998,Y 84.5628,Z 93,A 112.5337,B 24.9155,C -2.1221,E1 24.9261,E2 332.7251} C_DIS
LIN {X -42.1758,Y 86.1101,Z 93,A 110.6865,B 24.9148,C -2.1314,E1 24.9306,E2 334.5551} C_DIS
LIN {X -39.9293,Y 87.1754,Z 93,A 109.2034,B 24.9146,C -2.1338,E1 24.9344,E2 336.0363} C_DIS
LIN {X -37.7778,Y 88.129,Z 93,A 107.5953,B 24.915,C -2.1292,E1 24.9386,E2 337.6593} C_DIS
LIN {X -34.9843,Y 89.2729,Z 93,A 105.9125,B 24.9145,C -2.1357,E1 24.9429,E2 339.3302} C_DIS
LIN {X -32.3026,Y 90.2798,Z 93,A 104.2666,B 24.9141,C -2.14,E1 24.9472,E2 340.969} C_DIS
LIN {X -29.5909,Y 91.2027,Z 93,A 102.5077,B 24.9141,C -2.1406,E1 24.9518,E2 342.73} C_DIS
LIN {X -27.1959,Y 91.9453,Z 93,A 101.0483,B 24.9138,C -2.1435,E1 24.9557,E2 344.1848} C_DIS
LIN {X -24.9312,Y 92.585,Z 93,A 99.6389,B 24.9138,C -2.1449,E1 24.9595,E2 345.5932} C_DIS
LIN {X -22.6516,Y 93.169,Z 93,A 98.2292,B 24.9136,C -2.1461,E1 24.9633,E2 347.002} C_DIS
LIN {X -20.2907,Y 93.7116,Z 93,A 96.7123,B 24.9136,C -2.1451,E1 24.9675,E2 348.5233} C_DIS
LIN {X -17.0476,Y 94.3553,Z 93,A 94.7572,B 24.9136,C -2.1473,E1 24.9728,E2 350.4752} C_DIS
LIN {X -14.0692,Y 94.847,Z 93,A 92.7964,B 24.9138,C -2.1432,E1 24.9783,E2 352.4475} C_DIS
LIN {X -11.0764,Y 95.2411,Z 93,A 91.1015,B 24.9135,C -2.148,E1 24.983,E2 354.1321} C_DIS
LIN {X -8.2267,Y 95.5312,Z 93,A 89.3846,B 24.9135,C -2.1487,E1 24.9877,E2 355.8484} C_DIS
LIN {X -5.2153,Y 95.7411,Z 93,A 87.5824,B 24.9133,C -2.1495,E1 24.9927,E2 357.6493} C_DIS
LIN {X -2.3531,Y 95.8559,Z 93,A 85.9551,B 24.9131,C -2.1528,E1 24.9973,E2 359.2689} C_DIS
LIN {X 0.5112,Y 95.8817,Z 93,A 84.2046,B 24.9131,C -2.1519,E1 25.0022,E2 361.0216} C_DIS
LIN {X 3.5293,Y 95.8198,Z 93,A 82.2414,B 24.9136,C -2.1465,E1 25.0077,E2 362.9971} C_DIS
LIN {X 6.5437,Y 95.6595,Z 93,A 80.549,B 24.9133,C -2.1504,E1 25.0124,E2 364.6796} C_DIS
LIN {X 9.3984,Y 95.4231,Z 93,A 78.7261,B 24.9136,C -2.1464,E1 25.0175,E2 366.511} C_DIS
LIN {X 12.3973,Y 95.0782,Z 93,A 77.0342,B 24.9133,C -2.1499,E1 25.0221,E2 368.1932} C_DIS
LIN {X 15.7363,Y 94.5829,Z 93,A 75.0613,B 24.9133,C -2.1509,E1 25.0275,E2 370.1619} C_DIS
LIN {X 18.7062,Y 94.0424,Z 93,A 73.3017,B 24.9132,C -2.1517,E1 25.0324,E2 371.9176} C_DIS
LIN {X 21.0085,Y 93.555,Z 93,A 71.7005,B 24.9138,C -2.1441,E1 25.0368,E2 373.5346} C_DIS
LIN {X 23.9426,Y 92.8456,Z 93,A 70.0758,B 24.9134,C -2.1494,E1 25.0411,E2 375.1444} C_DIS
LIN {X 26.7058,Y 92.0907,Z 93,A 68.2397,B 24.9138,C -2.1438,E1 25.0461,E2 376.9908} C_DIS
LIN {X 29.5909,Y 91.2027,Z 93,A 66.5852,B 24.9135,C -2.1477,E1 25.0505,E2 378.6329} C_DIS
LIN {X 31.8203,Y 90.449,Z 93,A 65.1817,B 24.9135,C -2.1466,E1 25.0542,E2 380.0363} C_DIS
LIN {X 34.5085,Y 89.4598,Z 93,A 63.4736,B 24.9137,C -2.1451,E1 25.0586,E2 381.7443} C_DIS
LIN {X 36.6935,Y 88.586,Z 93,A 61.8742,B 24.9144,C -2.1367,E1 25.0628,E2 383.3598} C_DIS
LIN {X 39.4632,Y 87.3854,Z 93,A 60.1855,B 24.9142,C -2.1389,E1 25.0671,E2 385.0393} C_DIS
LIN {X 42.5146,Y 85.9422,Z 93,A 58.2164,B 24.9142,C -2.1382,E1 25.0721,E2 387.005} C_DIS
LIN {X 44.7475,Y 84.801,Z 93,A 56.7646,B 24.9142,C -2.1379,E1 25.0756,E2 388.4533} C_DIS
LIN {X 47.2614,Y 83.4281,Z 93,A 54.9381,B 24.9148,C -2.1313,E1 25.0801,E2 390.29} C_DIS
LIN {X 49.8633,Y 81.8975,Z 93,A 53.175,B 24.9148,C -2.1302,E1 25.0843,E2 392.0504} C_DIS
LIN {X 52.5179,Y 80.2216,Z 93,A 51.267,B 24.9152,C -2.1261,E1 25.0888,E2 393.9619} C_DIS
LIN {X 55.2112,Y 78.3939,Z 93,A 49.4528,B 24.9152,C -2.1276,E1 25.093,E2 395.7664} C_DIS
LIN {X 57.1185,Y 77.0154,Z 93,A 47.8557,B 24.9159,C -2.1182,E1 25.0966,E2 397.38} C_DIS
LIN {X 59.5135,Y 75.1778,Z 93,A 46.1696,B 24.9158,C -2.1192,E1 25.1003,E2 399.0574} C_DIS
LIN {X 62.1228,Y 73.0364,Z 93,A 44.2036,B 24.9159,C -2.1173,E1 25.1045,E2 401.0205} C_DIS
LIN {X 64.0114,Y 71.3869,Z 93,A 42.6689,B 24.9163,C -2.113,E1 25.1077,E2 402.5592} C_DIS
LIN {X 66.378,Y 69.1922,Z 93,A 40.7425,B 24.9166,C -2.1091,E1 25.1117,E2 404.4869} C_DIS
LIN {X 68.6277,Y 66.9637,Z 93,A 38.7547,B 24.9172,C -2.1015,E1 25.1156,E2 406.4842} C_DIS
LIN {X 70.7003,Y 64.7689,Z 93,A 37.1548,B 24.9169,C -2.1051,E1 25.1186,E2 408.0686} C_DIS
LIN {X 72.6048,Y 62.6293,Z 93,A 35.4518,B 24.9172,C -2.1015,E1 25.1217,E2 409.7724} C_DIS
LIN {X 74.4418,Y 60.4315,Z 93,A 33.7067,B 24.9176,C -2.0962,E1 25.1249,E2 411.5219} C_DIS
LIN {X 76.0193,Y 58.4348,Z 93,A 32.1616,B 24.918,C -2.0917,E1 25.1275,E2 413.0705} C_DIS
LIN {X 77.6482,Y 56.2543,Z 93,A 30.6139,B 24.918,C -2.0906,E1 25.1301,E2 414.6134} C_DIS
LIN {X 79.3522,Y 53.8218,Z 93,A 28.8113,B 24.9185,C -2.0851,E1 25.1329,E2 416.4201} C_DIS
LIN {X 81.0086,Y 51.2981,Z 93,A 27.0598,B 24.9187,C -2.0824,E1 25.1356,E2 418.1692} C_DIS
LIN {X 82.5032,Y 48.8546,Z 93,A 25.3063,B 24.9192,C -2.0763,E1 25.1381,E2 419.9281} C_DIS
LIN {X 84.0018,Y 46.2341,Z 93,A 23.3693,B 24.9199,C -2.0664,E1 25.1408,E2 421.8785} C_DIS
LIN {X 85.414,Y 43.5661,Z 93,A 21.7119,B 24.9199,C -2.067,E1 25.1429,E2 423.5257} C_DIS
LIN {X 86.8509,Y 40.6262,Z 93,A 19.7524,B 24.9203,C -2.0613,E1 25.1453,E2 425.488} C_DIS
LIN {X 88.129,Y 37.7778,Z 93,A 17.974,B 24.9205,C -2.0593,E1 25.1473,E2 427.2616} C_DIS
LIN {X 89.214,Y 35.1343,Z 93,A 16.2326,B 24.921,C -2.0531,E1 25.1491,E2 429.0079} C_DIS
LIN {X 90.2798,Y 32.3026,Z 93,A 14.2648,B 24.9218,C -2.0416,E1 25.151,E2 430.9917} C_DIS
LIN {X 91.2502,Y 29.4441,Z 93,A 12.6885,B 24.9216,C -2.0449,E1 25.1524,E2 432.5513} C_DIS
LIN {X 92.0907,Y 26.7058,Z 93,A 10.9881,B 24.922,C -2.0402,E1 25.1537,E2 434.2532} C_DIS
LIN {X 92.8456,Y 23.9426,Z 93,A 9.2456,B 24.9224,C -2.0338,E1 25.155,E2 436.0008} C_DIS
LIN {X 93.4399,Y 21.5065,Z 93,A 7.7147,B 24.9229,C -2.0279,E1 25.156,E2 437.5366} C_DIS
LIN {X 94.139,Y 18.2042,Z 93,A 5.7555,B 24.9232,C -2.0239,E1 25.1571,E2 439.4939} C_DIS
LIN {X 94.5829,Y 15.7363,Z 93,A 4.2228,B 24.9236,C -2.0179,E1 25.1578,E2 441.0318} C_DIS
LIN {X 95.0612,Y 12.5285,Z 93,A 2.297,B 24.9241,C -2.0123,E1 25.1586,E2 442.9596} C_DIS
LIN {X 95.4231,Y 9.3983,Z 93,A 0.3176,B 24.9248,C -2.0026,E1 25.1592,E2 444.9502} C_DIS
LIN {X 95.6699,Y 6.3898,Z 93,A -1.3636,B 24.9248,C -2.0015,E1 25.1595,E2 446.6238} C_DIS
LIN {X 95.8355,Y 3.0183,Z 93,A -3.3241,B 24.9252,C -1.9972,E1 25.1597,E2 448.5827} C_DIS
LIN {X 95.8851,Y 0.1467,Z 93,A -5.0448,B 24.9256,C -1.9915,E1 25.1597,E2 450.3067} C_DIS
LIN {X 95.8355,Y -3.0183,Z 93,A -6.8646,B 24.9259,C -1.9882,E1 25.1597,E2 452.1234} C_DIS
LIN {X 95.7043,Y -5.8797,Z 93,A -8.5641,B 24.9263,C -1.9832,E1 25.1594,E2 453.8248} C_DIS
LIN {X 95.4842,Y -8.7357,Z 93,A -10.3061,B 24.9268,C -1.9765,E1 25.159,E2 455.5722} C_DIS
LIN {X 95.1637,Y -11.7373,Z 93,A -12.2564,B 24.9276,C -1.965,E1 25.1584,E2 457.538} C_DIS
LIN {X 94.7453,Y -14.7269,Z 93,A -13.9233,B 24.9276,C -1.9645,E1 25.1577,E2 459.1962} C_DIS
LIN {X 94.2649,Y -17.5507,Z 93,A -15.7412,B 24.9283,C -1.955,E1 25.1568,E2 461.0262} C_DIS
LIN {X 93.6639,Y -20.509,Z 93,A -17.4223,B 24.9284,C -1.9539,E1 25.1558,E2 462.6999} C_DIS
LIN {X 93.0112,Y -23.2981,Z 93,A -19.0375,B 24.9285,C -1.9522,E1 25.1548,E2 464.3099} C_DIS
LIN {X 92.4115,Y -25.5737,Z 93,A -20.434,B 24.9288,C -1.9481,E1 25.1538,E2 465.7079} C_DIS
LIN {X 91.756,Y -27.8339,Z 93,A -21.8306,B 24.9291,C -1.9441,E1 25.1527,E2 467.1061} C_DIS
LIN {X 90.9621,Y -30.3241,Z 93,A -23.5105,B 24.9298,C -1.9347,E1 25.1512,E2 468.7986} C_DIS
LIN {X 89.8766,Y -33.4081,Z 93,A -25.449,B 24.9302,C -1.9292,E1 25.1494,E2 470.7392} C_DIS
LIN {X 88.7787,Y -36.22,Z 93,A -27.1993,B 24.9305,C -1.9257,E1 25.1475,E2 472.4879} C_DIS
LIN {X 87.6588,Y -38.8565,Z 93,A -29.0098,B 24.9311,C -1.9167,E1 25.1455,E2 474.3099} C_DIS
LIN {X 86.3906,Y -41.5959,Z 93,A -30.607,B 24.9309,C -1.9192,E1 25.1436,E2 475.8925} C_DIS
LIN {X 85.3438,Y -43.7035,Z 93,A -32.004,B 24.9312,C -1.9154,E1 25.1419,E2 477.291} C_DIS
LIN {X 84.0018,Y -46.2341,Z 93,A -33.9002,B 24.9321,C -1.9033,E1 25.1393,E2 479.2059} C_DIS
LIN {X 82.5032,Y -48.8546,Z 93,A -35.5823,B 24.9321,C -1.9028,E1 25.137,E2 480.8806} C_DIS
LIN {X 80.7325,Y -51.7283,Z 93,A -37.5444,B 24.9324,C -1.8991,E1 25.1341,E2 482.8414} C_DIS
LIN {X 79.3522,Y -53.8218,Z 93,A -39.0764,B 24.9328,C -1.8937,E1 25.1317,E2 484.3787} C_DIS
LIN {X 77.7105,Y -56.1691,Z 93,A -40.8883,B 24.9334,C -1.8851,E1 25.1287,E2 486.2019} C_DIS
LIN {X 75.9025,Y -58.5864,Z 93,A -42.4862,B 24.9332,C -1.8881,E1 25.1261,E2 487.7852} C_DIS
LIN {X 74.4418,Y -60.4315,Z 93,A -43.8844,B 24.9334,C -1.8847,E1 25.1236,E2 489.185} C_DIS
LIN {X 72.6048,Y -62.6293,Z 93,A -45.5862,B 24.9337,C -1.8806,E1 25.1205,E2 490.8886} C_DIS
LIN {X 70.7003,Y -64.7689,Z 93,A -47.331,B 24.9341,C -1.875,E1 25.1173,E2 492.6388} C_DIS
LIN {X 68.6277,Y -66.9637,Z 93,A -49.2316,B 24.9347,C -1.8668,E1 25.1136,E2 494.5505} C_DIS
LIN {X 66.4845,Y -69.0895,Z 93,A -50.9603,B 24.9347,C -1.8654,E1 25.1101,E2 496.2755} C_DIS
LIN {X 64.0114,Y -71.3869,Z 93,A -52.9264,B 24.935,C -1.8626,E1 25.1061,E2 498.2403} C_DIS
LIN {X 62.1228,Y -73.0364,Z 93,A -54.46,B 24.9353,C -1.8578,E1 25.1028,E2 499.7791} C_DIS
LIN {X 59.9145,Y -74.8608,Z 93,A -56.0784,B 24.9353,C -1.8575,E1 25.0993,E2 501.392} C_DIS
LIN {X 58.0593,Y -76.3087,Z 93,A -57.6739,B 24.936,C -1.8474,E1 25.0958,E2 503.0055} C_DIS
LIN {X 55.6274,Y -78.097,Z 93,A -59.3591,B 24.936,C -1.8482,E1 25.092,E2 504.683} C_DIS
LIN {X 52.844,Y -80.0067,Z 93,A -61.3247,B 24.9361,C -1.8461,E1 25.0874,E2 506.6471} C_DIS
LIN {X 50.7337,Y -81.3612,Z 93,A -62.7746,B 24.9361,C -1.845,E1 25.084,E2 508.0947} C_DIS
LIN {X 48.2817,Y -82.8419,Z 93,A -64.6752,B 24.9369,C -1.8348,E1 25.0794,E2 510.0136} C_DIS
LIN {X 45.6491,Y -84.3191,Z 93,A -66.2674,B 24.9366,C -1.8395,E1 25.0755,E2 511.59} C_DIS
LIN {X 43.1109,Y -85.6466,Z 93,A -68.1775,B 24.9373,C -1.8293,E1 25.0707,E2 513.519} C_DIS
LIN {X 40.3927,Y -86.9597,Z 93,A -69.8647,B 24.9372,C -1.8308,E1 25.0665,E2 515.1985} C_DIS
LIN {X 37.7778,Y -88.129,Z 93,A -71.6814,B 24.9376,C -1.8243,E1 25.0618,E2 517.026} C_DIS
LIN {X 34.9843,Y -89.2729,Z 93,A -73.369,B 24.9375,C -1.8261,E1 25.0575,E2 518.7057} C_DIS
LIN {X 32.3026,Y -90.2798,Z 93,A -74.9907,B 24.9375,C -1.8271,E1 25.0532,E2 520.3216} C_DIS
LIN {X 30.0773,Y -91.0453,Z 93,A -76.3929,B 24.9375,C -1.8255,E1 25.0495,E2 521.7249} C_DIS
LIN {X 27.3188,Y -91.9088,Z 93,A -78.1506,B 24.9378,C -1.8224,E1 25.0448,E2 523.4867} C_DIS
LIN {X 24.4377,Y -92.7183,Z 93,A -80.0868,B 24.9383,C -1.8151,E1 25.0396,E2 525.4372} C_DIS
LIN {X 21.5066,Y -93.4399,Z 93,A -81.7852,B 24.9381,C -1.8172,E1 25.035,E2 527.1282} C_DIS
LIN {X 18.7062,Y -94.0424,Z 93,A -83.6047,B 24.9385,C -1.8117,E1 25.03,E2 528.9582} C_DIS
LIN {X 15.7363,Y -94.5829,Z 93,A -85.2948,B 24.9383,C -1.8145,E1 25.0253,E2 530.6401} C_DIS
LIN {X 12.9042,Y -95.0125,Z 93,A -86.9183,B 24.9382,C -1.8164,E1 25.0209,E2 532.2575} C_DIS
LIN {X 10.0602,Y -95.3538,Z 93,A -88.6705,B 24.9383,C -1.814,E1 25.016,E2 534.0142} C_DIS
LIN {X 7.5633,Y -95.5843,Z 93,A -90.2101,B 24.9385,C -1.8117,E1 25.0117,E2 535.5582} C_DIS
LIN {X 4.7048,Y -95.7693,Z 93,A -92.031,B 24.9388,C -1.8071,E1 25.0066,E2 537.3895} C_DIS
LIN {X 1.6878,Y -95.8682,Z 93,A -93.6378,B 24.9384,C -1.8136,E1 25.0022,E2 538.9806} C_DIS
LIN {X 1.6878,Y -95.8682,Z 93,A -93.6378,B 24.9384,C -1.8136,E1 25.0022,E2 538.9806} C_DIS
Enddeposition()
LIN {X 0.6414,Y -94.9343,Z 93,A -93.7272,B 24.9359,C -1.849,E1 25.0022,E2 538.9861} C_DIS
Startdeposition()
$VEL.CP = VEL_PRINT
LIN {X 3.4097,Y -94.8782,Z 93,A -91.8242,B 24.9353,C -1.8577,E1 25.0075,E2 537.0627} C_DIS
LIN {X 6.3349,Y -94.7266,Z 93,A -89.9772,B 24.9351,C -1.8613,E1 25.0127,E2 535.2079} C_DIS
LIN {X 9.976,Y -94.4126,Z 93,A -87.6701,B 24.9347,C -1.8662,E1 25.0191,E2 532.8907} C_DIS
LIN {X 14.0588,Y -93.8925,Z 93,A -85.3485,B 24.935,C -1.862,E1 25.0255,E2 530.5811} C_DIS
LIN {X 17.4365,Y -93.3247,Z 93,A -83.1614,B 24.9346,C -1.868,E1 25.0315,E2 528.3823} C_DIS
LIN {X 21.8583,Y -92.389,Z 93,A -80.5,B 24.9346,C -1.868,E1 25.0388,E2 525.7241} C_DIS
LIN {X 26.5746,Y -91.1441,Z 93,A -77.8555,B 24.9351,C -1.8603,E1 25.0459,E2 523.1022} C_DIS
LIN {X 29.2623,Y -90.3159,Z 93,A -75.9172,B 24.9344,C -1.8712,E1 25.0511,E2 521.1419} C_DIS
LIN {X 32.488,Y -89.2064,Z 93,A -73.9005,B 24.9343,C -1.8723,E1 25.0564,E2 519.1266} C_DIS
LIN {X 35.9577,Y -87.8654,Z 93,A -71.6386,B 24.934,C -1.876,E1 25.0623,E2 516.8609} C_DIS
LIN {X 39.25,Y -86.4451,Z 93,A -69.6143,B 24.9342,C -1.8741,E1 25.0674,E2 514.846} C_DIS
LIN {X 42.1326,Y -85.077,Z 93,A -67.6289,B 24.9338,C -1.8795,E1 25.0724,E2 512.8532} C_DIS
LIN {X 44.6649,Y -83.7767,Z 93,A -65.0628,B 24.9313,C -1.9141,E1 25.0789,E2 510.2125} C_DIS
LIN {X 48.7221,Y -81.484,Z 93,A -63.0624,B 24.9331,C -1.8887,E1 25.0836,E2 508.2782} C_DIS
LIN {X 51.4968,Y -79.7583,Z 93,A -61.056,B 24.9328,C -1.8938,E1 25.0883,E2 506.2663} C_DIS
LIN {X 53.9029,Y -78.1527,Z 93,A -59.0106,B 24.9317,C -1.9086,E1 25.0931,E2 504.1929} C_DIS
LIN {X 57.998,Y -75.1631,Z 93,A -56.4005,B 24.9325,C -1.8981,E1 25.0988,E2 501.6171} C_DIS
LIN {X 60.481,Y -73.1804,Z 93,A -54.437,B 24.932,C -1.904,E1 25.1031,E2 499.6469} C_DIS
LIN {X 63.0443,Y -70.9845,Z 93,A -52.5216,B 24.932,C -1.904,E1 25.1071,E2 497.739} C_DIS
LIN {X 65.3248,Y -68.8917,Z 93,A -50.3877,B 24.931,C -1.9186,E1 25.1115,E2 495.5796} C_DIS
LIN {X 68.0228,Y -66.2297,Z 93,A -48.1932,B 24.9308,C -1.9206,E1 25.1158,E2 493.3896} C_DIS
LIN {X 70.6128,Y -63.4595,Z 93,A -46.3482,B 24.9316,C -1.9096,E1 25.1193,E2 491.5788} C_DIS
LIN {X 72.496,Y -61.3001,Z 93,A -43.6313,B 24.9286,C -1.9517,E1 25.1243,E2 488.7747} C_DIS
LIN {X 75.0108,Y -58.1956,Z 93,A -41.8972,B 24.93,C -1.9322,E1 25.1272,E2 487.0949} C_DIS
LIN {X 77.0336,Y -55.4911,Z 93,A -39.8959,B 24.9297,C -1.9363,E1 25.1305,E2 485.0935} C_DIS
LIN {X 80.3428,Y -50.5805,Z 93,A -36.3036,B 24.9289,C -1.947,E1 25.1361,E2 481.4938} C_DIS
LIN {X 82.0513,Y -47.761,Z 93,A -34.1717,B 24.9281,C -1.9582,E1 25.1391,E2 479.3465} C_DIS
LIN {X 83.7957,Y -44.6287,Z 93,A -32.2326,B 24.9283,C -1.9559,E1 25.1417,E2 477.423} C_DIS
LIN {X 85.0847,Y -42.1171,Z 93,A -30.4554,B 24.9277,C -1.9638,E1 25.1439,E2 475.6365} C_DIS
LIN {X 86.4485,Y -39.2425,Z 93,A -28.3011,B 24.9266,C -1.9786,E1 25.1465,E2 473.459} C_DIS
LIN {X 88.4748,Y -34.4318,Z 93,A -25.5119,B 24.9269,C -1.9743,E1 25.1494,E2 470.6953} C_DIS
LIN {X 89.3071,Y -32.212,Z 93,A -23.8642,B 24.926,C -1.9871,E1 25.151,E2 469.0266} C_DIS
LIN {X 90.6761,Y -28.1263,Z 93,A -21.5303,B 24.9261,C -1.9849,E1 25.153,E2 466.711} C_DIS
LIN {X 91.5633,Y -25.0904,Z 93,A -19.6048,B 24.9256,C -1.9916,E1 25.1545,E2 464.7809} C_DIS
LIN {X 92.3341,Y -22.0873,Z 93,A -17.6869,B 24.9251,C -1.9993,E1 25.1557,E2 462.8559} C_DIS
LIN {X 92.9746,Y -19.2089,Z 93,A -15.9208,B 24.9247,C -2.0045,E1 25.1568,E2 461.0878} C_DIS
LIN {X 93.7451,Y -15.0124,Z 93,A -13.2883,B 24.9239,C -2.0149,E1 25.158,E2 458.4461} C_DIS
LIN {X 94.254,Y -11.3823,Z 93,A -11.1212,B 24.9235,C -2.0203,E1 25.1588,E2 456.2791} C_DIS
LIN {X 94.5859,Y -8.1881,Z 93,A -9.1586,B 24.9229,C -2.0275,E1 25.1593,E2 454.3113} C_DIS
LIN {X 94.8287,Y -4.5845,Z 93,A -6.9916,B 24.9224,C -2.034,E1 25.1597,E2 452.1417} C_DIS
LIN {X 94.9261,Y -1.5263,Z 93,A -5.2362,B 24.9222,C -2.0364,E1 25.1597,E2 450.3911} C_DIS
LIN {X 94.9113,Y 2.3311,Z 93,A -2.8146,B 24.9214,C -2.0475,E1 25.1597,E2 447.9577} C_DIS
LIN {X 94.7371,Y 6.1793,Z 93,A -0.6187,B 24.9212,C -2.05,E1 25.1593,E2 445.769} C_DIS
LIN {X 94.4951,Y 9.1723,Z 93,A 1.38,B 24.9202,C -2.0629,E1 25.1588,E2 443.7517} C_DIS
LIN {X 94.0113,Y 13.2343,Z 93,A 3.629,B 24.9202,C -2.0622,E1 25.158,E2 441.5175} C_DIS
LIN {X 93.4878,Y 16.5337,Z 93,A 5.7159,B 24.9195,C -2.0713,E1 25.157,E2 439.4216} C_DIS
LIN {X 92.207,Y 22.6084,Z 93,A 9.3666,B 24.9189,C -2.0791,E1 25.1549,E2 435.7735} C_DIS
LIN {X 91.3401,Y 25.889,Z 93,A 11.1855,B 24.9191,C -2.0766,E1 25.1535,E2 433.971} C_DIS
LIN {X 89.7636,Y 30.92,Z 93,A 14.6703,B 24.9175,C -2.0976,E1 25.1505,E2 430.4563} C_DIS
LIN {X 88.4905,Y 34.3918,Z 93,A 16.5444,B 24.918,C -2.0906,E1 25.1487,E2 428.6094} C_DIS
LIN {X 87.2985,Y 37.3157,Z 93,A 18.702,B 24.9168,C -2.1056,E1 25.1464,E2 426.428} C_DIS
LIN {X 85.9058,Y 40.4178,Z 93,A 20.6297,B 24.9168,C -2.1067,E1 25.1441,E2 424.5082} C_DIS
LIN {X 84.4858,Y 43.3061,Z 93,A 22.5703,B 24.9163,C -2.1121,E1 25.1417,E2 422.5653} C_DIS
LIN {X 83.2838,Y 45.5762,Z 93,A 24.408,B 24.9151,C -2.1272,E1 25.1392,E2 420.7016} C_DIS
LIN {X 81.1096,Y 49.3405,Z 93,A 26.5217,B 24.9161,C -2.1149,E1 25.1363,E2 418.6278} C_DIS
LIN {X 78.9152,Y 52.7819,Z 93,A 29.2537,B 24.9148,C -2.1313,E1 25.1321,E2 415.8706} C_DIS
LIN {X 76.967,Y 55.5844,Z 93,A 31.2667,B 24.9145,C -2.1347,E1 25.1288,E2 413.8594} C_DIS
LIN {X 74.7717,Y 58.5035,Z 93,A 33.4633,B 24.9141,C -2.1398,E1 25.1251,E2 411.6613} C_DIS
LIN {X 72.6032,Y 61.1743,Z 93,A 35.3729,B 24.9142,C -2.1384,E1 25.1217,E2 409.7638} C_DIS
LIN {X 69.3102,Y 64.8798,Z 93,A 38.9842,B 24.9118,C -2.1683,E1 25.1148,E2 406.0978} C_DIS
LIN {X 66.9626,Y 67.3007,Z 93,A 40.2713,B 24.9137,C -2.1447,E1 25.1124,E2 404.8718} C_DIS
LIN {X 64.7675,Y 69.4159,Z 93,A 42.3019,B 24.9128,C -2.1556,E1 25.1083,E2 402.824} C_DIS
LIN {X 62.5066,Y 71.4575,Z 93,A 44.2586,B 24.9122,C -2.1636,E1 25.1042,E2 400.8561} C_DIS
LIN {X 60.6575,Y 73.0337,Z 93,A 46.6154,B 24.9093,C -2.1995,E1 25.0989,E2 398.4233} C_DIS
LIN {X 56.6148,Y 76.2121,Z 93,A 48.8214,B 24.9115,C -2.1717,E1 25.0942,E2 396.2913} C_DIS
LIN {X 53.7877,Y 78.2328,Z 93,A 51.152,B 24.9106,C -2.1837,E1 25.0888,E2 393.9401} C_DIS
LIN {X 50.3673,Y 80.476,Z 93,A 53.2511,B 24.9113,C -2.1741,E1 25.0839,E2 391.8706} C_DIS
LIN {X 47.5118,Y 82.1945,Z 93,A 55.7208,B 24.9097,C -2.1937,E1 25.0779,E2 389.362} C_DIS
LIN {X 44.7082,Y 83.7538,Z 93,A 57.2424,B 24.9108,C -2.1812,E1 25.0742,E2 387.8743} C_DIS
LIN {X 41.8941,Y 85.1952,Z 93,A 59.1279,B 24.9106,C -2.1828,E1 25.0695,E2 385.9902} C_DIS
LIN {X 38.9398,Y 86.5849,Z 93,A 61.237,B 24.91,C -2.1901,E1 25.0641,E2 383.869} C_DIS
LIN {X 35.2256,Y 88.163,Z 93,A 63.6249,B 24.91,C -2.1909,E1 25.058,E2 381.4848} C_DIS
LIN {X 32.6412,Y 89.1505,Z 93,A 65.5131,B 24.9092,C -2.2003,E1 25.053,E2 379.5783} C_DIS
LIN {X 29.5688,Y 90.2168,Z 93,A 67.4191,B 24.9092,C -2.1999,E1 25.0479,E2 377.677} C_DIS
LIN {X 25.5038,Y 91.4492,Z 93,A 69.7819,B 24.9097,C -2.1945,E1 25.0416,E2 375.3309} C_DIS
LIN {X 20.0256,Y 92.8023,Z 93,A 73.3372,B 24.9091,C -2.2017,E1 25.0319,E2 371.7637} C_DIS
LIN {X 15.8616,Y 93.604,Z 93,A 75.5127,B 24.9101,C -2.1891,E1 25.0261,E2 369.6204} C_DIS
LIN {X 11.8554,Y 94.1956,Z 93,A 78.1092,B 24.9096,C -2.195,E1 25.0188,E2 367.012} C_DIS
LIN {X 9.1995,Y 94.4926,Z 93,A 79.8558,B 24.9092,C -2.1999,E1 25.014,E2 365.2549} C_DIS
LIN {X 5.5166,Y 94.7781,Z 93,A 81.9852,B 24.9095,C -2.1965,E1 25.0081,E2 363.1346} C_DIS
LIN {X 1.9725,Y 94.9179,Z 93,A 84.0812,B 24.9096,C -2.1947,E1 25.0022,E2 361.0433} C_DIS
LIN {X -2.1149,Y 94.9153,Z 93,A 86.6635,B 24.9094,C -2.1982,E1 24.995,E2 358.4528} C_DIS
LIN {X -5.8508,Y 94.7592,Z 93,A 88.8855,B 24.9095,C -2.1961,E1 24.9888,E2 356.235} C_DIS
LIN {X -8.5708,Y 94.5506,Z 93,A 90.8521,B 24.9087,C -2.2064,E1 24.9833,E2 354.243} C_DIS
LIN {X -13.6132,Y 93.9574,Z 93,A 94.1117,B 24.9083,C -2.2112,E1 24.9742,E2 350.9695} C_DIS
LIN {X -17.2702,Y 93.3553,Z 93,A 95.8502,B 24.9098,C -2.1924,E1 24.9695,E2 349.2738} C_DIS
LIN {X -20.5865,Y 92.68,Z 93,A 97.8102,B 24.9102,C -2.1879,E1 24.9642,E2 347.3222} C_DIS
LIN {X -25.4358,Y 91.4685,Z 93,A 100.879,B 24.9103,C -2.1866,E1 24.9559,E2 344.2519} C_DIS
LIN {X -28.3809,Y 90.5972,Z 93,A 102.582,B 24.9109,C -2.1795,E1 24.9514,E2 342.563} C_DIS
LIN {X -32.7762,Y 89.1013,Z 93,A 105.585,B 24.9106,C -2.1827,E1 24.9435,E2 339.5464} C_DIS
LIN {X -35.9074,Y 87.8858,Z 93,A 107.5515,B 24.911,C -2.1779,E1 24.9384,E2 337.5871} C_DIS
LIN {X -38.8599,Y 86.6209,Z 93,A 109.5147,B 24.9112,C -2.1759,E1 24.9333,E2 335.624} C_DIS
LIN {X -42.5001,Y 84.8948,Z 93,A 112.0024,B 24.9114,C -2.1739,E1 24.9271,E2 333.1346} C_DIS
LIN {X -45.8216,Y 83.1498,Z 93,A 114.1832,B 24.9119,C -2.1673,E1 24.9218,E2 330.9633} C_DIS
LIN {X -48.2508,Y 81.7626,Z 93,A 115.8634,B 24.9122,C -2.1641,E1 24.9177,E2 329.2858} C_DIS
LIN {X -51.2124,Y 79.9409,Z 93,A 118.0841,B 24.9122,C -2.1641,E1 24.9124,E2 327.0579} C_DIS
LIN {X -54.6651,Y 77.6228,Z 93,A 120.4021,B 24.9131,C -2.1529,E1 24.9071,E2 324.7589} C_DIS
LIN {X -58.1199,Y 75.0691,Z 93,A 123.0086,B 24.9135,C -2.148,E1 24.9013,E2 322.1548} C_DIS
LIN {X -61.5963,Y 72.2437,Z 93,A 125.9034,B 24.9135,C -2.1483,E1 24.8951,E2 319.2484} C_DIS
LIN {X -63.8408,Y 70.2696,Z 93,A 127.8067,B 24.9135,C -2.1473,E1 24.8911,E2 317.3397} C_DIS
LIN {X -65.9739,Y 68.2694,Z 93,A 129.7083,B 24.9135,C -2.1476,E1 24.8873,E2 315.4295} C_DIS
LIN {X -68.9389,Y 65.2747,Z 93,A 132.0711,B 24.9145,C -2.1356,E1 24.8827,E2 313.0852} C_DIS
LIN {X -71.2946,Y 62.6932,Z 93,A 134.1235,B 24.915,C -2.1284,E1 24.8789,E2 311.0408} C_DIS
LIN {X -73.2611,Y 60.3838,Z 93,A 135.9583,B 24.9154,C -2.1238,E1 24.8756,E2 309.2084} C_DIS
LIN {X -75.1654,Y 57.995,Z 93,A 137.8762,B 24.9156,C -2.1213,E1 24.8723,E2 307.2875} C_DIS
LIN {X -76.8524,Y 55.7417,Z 93,A 139.6547,B 24.9158,C -2.1193,E1 24.8694,E2 305.5053} C_DIS
LIN {X -78.8593,Y 52.8645,Z 93,A 141.7644,B 24.9163,C -2.1132,E1 24.8661,E2 303.3996} C_DIS
LIN {X -80.9109,Y 49.6675,Z 93,A 143.9127,B 24.9171,C -2.1021,E1 24.8629,E2 301.2667} C_DIS
LIN {X -82.5953,Y 46.8142,Z 93,A 146.4845,B 24.9161,C -2.1147,E1 24.8593,E2 298.6516} C_DIS
LIN {X -84.2273,Y 43.8092,Z 93,A 148.2123,B 24.9175,C -2.0978,E1 24.8571,E2 296.9547} C_DIS
LIN {X -85.9847,Y 40.2483,Z 93,A 150.4517,B 24.9184,C -2.0857,E1 24.8544,E2 294.7321} C_DIS
LIN {X -87.8,Y 36.1183,Z 93,A 153.2189,B 24.919,C -2.0789,E1 24.8513,E2 291.9659} C_DIS
LIN {X -88.9054,Y 33.3046,Z 93,A 155.01,B 24.9195,C -2.0723,E1 24.8495,E2 290.1806} C_DIS
LIN {X -89.9463,Y 30.3795,Z 93,A 156.8408,B 24.92,C -2.0651,E1 24.8479,E2 288.3564} C_DIS
LIN {X -91.3265,Y 25.937,Z 93,A 160.338,B 24.919,C -2.0782,E1 24.8451,E2 284.8077} C_DIS
LIN {X -92.268,Y 22.3582,Z 93,A 161.9042,B 24.9212,C -2.05,E1 24.8441,E2 283.2998} C_DIS
LIN {X -93.7138,Y 15.2044,Z 93,A 166.8627,B 24.9209,C -2.0534,E1 24.8415,E2 278.3038} C_DIS
LIN {X -94.51,Y 9.0107,Z 93,A 170.7421,B 24.9216,C -2.0448,E1 24.8403,E2 274.4216} C_DIS
LIN {X -94.774,Y 5.5907,Z 93,A 172.3909,B 24.9231,C -2.0248,E1 24.84,E2 272.8108} C_DIS
LIN {X -94.9193,Y 1.8972,Z 93,A 174.5467,B 24.9238,C -2.0153,E1 24.8398,E2 270.6647} C_DIS
LIN {X -94.9268,Y -1.4878,Z 93,A 176.4403,B 24.9247,C -2.004,E1 24.8398,E2 268.7866} C_DIS
LIN {X -94.7058,Y -6.6424,Z 93,A 179.8197,B 24.9248,C -2.0024,E1 24.8403,E2 265.3906} C_DIS
LIN {X -94.0808,Y -12.7415,Z 93,A -176.439,B 24.9256,C -1.992,E1 24.8415,E2 261.6517} C_DIS
LIN {X -93.5362,Y -16.2643,Z 93,A -174.2694,B 24.9261,C -1.9858,E1 24.8425,E2 259.4839} C_DIS
LIN {X -92.9059,Y -19.5438,Z 93,A -172.3373,B 24.9267,C -1.9769,E1 24.8435,E2 257.5617} C_DIS
LIN {X -92.1987,Y -22.6423,Z 93,A -170.4391,B 24.9272,C -1.9704,E1 24.8447,E2 255.6679} C_DIS
LIN {X -91.3888,Y -25.7169,Z 93,A -168.4993,B 24.9276,C -1.9653,E1 24.8462,E2 253.7292} C_DIS
LIN {X -90.5289,Y -28.6011,Z 93,A -166.6029,B 24.9278,C -1.9624,E1 24.8477,E2 251.8287} C_DIS
LIN {X -89.7189,Y -31.0474,Z 93,A -165.077,B 24.9282,C -1.9568,E1 24.8491,E2 250.3073} C_DIS
LIN {X -88.753,Y -33.7071,Z 93,A -162.3057,B 24.926,C -1.9863,E1 24.852,E2 247.4503} C_DIS
LIN {X -86.7189,Y -38.6423,Z 93,A -160.3288,B 24.9297,C -1.9367,E1 24.854,E2 245.5806} C_DIS
LIN {X -85.3125,Y -41.6574,Z 93,A -158.0592,B 24.9295,C -1.9395,E1 24.8568,E2 243.2922} C_DIS
LIN {X -83.9095,Y -44.4127,Z 93,A -156.1014,B 24.9296,C -1.9373,E1 24.8593,E2 241.3289} C_DIS
LIN {X -82.0831,Y -47.7057,Z 93,A -154.051,B 24.9306,C -1.9241,E1 24.8621,E2 239.2995} C_DIS
LIN {X -79.1341,Y -52.4509,Z 93,A -150.4767,B 24.9308,C -1.9218,E1 24.8675,E2 235.7124} C_DIS
LIN {X -77.409,Y -54.965,Z 93,A -148.6884,B 24.9312,C -1.9156,E1 24.8703,E2 233.9303} C_DIS
LIN {X -75.3249,Y -57.7879,Z 93,A -146.4928,B 24.9314,C -1.913,E1 24.874,E2 231.7304} C_DIS
LIN {X -72.887,Y -60.834,Z 93,A -144.0787,B 24.9317,C -1.9094,E1 24.8783,E2 229.3135} C_DIS
LIN {X -70.6762,Y -63.3887,Z 93,A -142.271,B 24.9325,C -1.8972,E1 24.8816,E2 227.5267} C_DIS
LIN {X -68.5596,Y -65.6728,Z 93,A -140.2801,B 24.9325,C -1.8968,E1 24.8854,E2 225.5282} C_DIS
LIN {X -66.466,Y -67.7912,Z 93,A -138.4614,B 24.9328,C -1.8937,E1 24.889,E2 223.7091} C_DIS
LIN {X -64.3146,Y -69.8349,Z 93,A -136.5747,B 24.9328,C -1.8932,E1 24.8928,E2 221.8158} C_DIS
LIN {X -60.1722,Y -73.4357,Z 93,A -132.8196,B 24.9322,C -1.9017,E1 24.9009,E2 218.0261} C_DIS
LIN {X -57.5272,Y -75.5258,Z 93,A -131.2972,B 24.9337,C -1.8809,E1 24.9042,E2 216.5476} C_DIS
LIN {X -55.0917,Y -77.3186,Z 93,A -129.394,B 24.9337,C -1.8804,E1 24.9085,E2 214.6388} C_DIS
LIN {X -52.477,Y -79.1169,Z 93,A -127.4545,B 24.9339,C -1.8782,E1 24.913,E2 212.6982} C_DIS
LIN {X -49.9132,Y -80.7597,Z 93,A -125.0025,B 24.9326,C -1.8963,E1 24.919,E2 210.1956} C_DIS
LIN {X -46.5017,Y -82.7702,Z 93,A -123.2879,B 24.9345,C -1.87,E1 24.923,E2 208.5385} C_DIS
LIN {X -43.5819,Y -84.3448,Z 93,A -121.2132,B 24.9345,C -1.8698,E1 24.9281,E2 206.4584} C_DIS
LIN {X -40.1276,Y -86.0409,Z 93,A -118.896,B 24.9347,C -1.8669,E1 24.9339,E2 204.1422} C_DIS
LIN {X -36.7791,Y -87.5246,Z 93,A -116.7959,B 24.9351,C -1.8608,E1 24.9393,E2 202.0517} C_DIS
LIN {X -32.5587,Y -89.1806,Z 93,A -113.5696,B 24.9341,C -1.8751,E1 24.9478,E2 198.7845} C_DIS
LIN {X -28.0635,Y -90.6956,Z 93,A -111.273,B 24.9356,C -1.8533,E1 24.9538,E2 196.5356} C_DIS
LIN {X -23.3595,Y -92.0199,Z 93,A -108.106,B 24.9352,C -1.859,E1 24.9624,E2 193.3502} C_DIS
LIN {X -19.8616,Y -92.8381,Z 93,A -105.9414,B 24.9352,C -1.8578,E1 24.9683,E2 191.1856} C_DIS
LIN {X -17.2935,Y -93.3511,Z 93,A -104.2281,B 24.935,C -1.8619,E1 24.973,E2 189.4609} C_DIS
LIN {X -13.4182,Y -93.9851,Z 93,A -102.1493,B 24.9358,C -1.8511,E1 24.9787,E2 187.4059} C_DIS
LIN {X -10.4611,Y -94.3614,Z 93,A -100.125,B 24.9352,C -1.8587,E1 24.9844,E2 185.3621} C_DIS
LIN {X -6.7642,Y -94.6975,Z 93,A -98.0161,B 24.9356,C -1.854,E1 24.9902,E2 183.2635} C_DIS
LIN {X -4.5292,Y -94.8311,Z 93,A -96.7669,B 24.9358,C -1.8505,E1 24.9937,E2 182.0223} C_DIS
LIN {X -1.4739,Y -94.9271,Z 93,A -94.7438,B 24.9353,C -1.8571,E1 24.9994,E2 179.9832} C_DIS
LIN {X -1.4739,Y -94.9271,Z 93,A -94.7438,B 24.9353,C -1.8571,E1 24.9994,E2 179.9832} C_DIS
Enddeposition()
LIN {X 0.6292,Y -93.9891,Z 93,A -93.6795,B 24.9347,C -1.8665,E1 25.0024,E2 178.8967} C_DIS
Startdeposition()
$VEL.CP = VEL_PRINT
LIN {X -2.5353,Y -93.9597,Z 93,A -96.5964,B 24.9371,C -1.8318,E1 24.994,E2 181.8962} C_DIS
LIN {X -5.8145,Y -93.8147,Z 93,A -98.4408,B 24.9367,C -1.837,E1 24.9889,E2 183.7286} C_DIS
LIN {X -9.1654,Y -93.5468,Z 93,A -100.8417,B 24.9376,C -1.8251,E1 24.9821,E2 186.159} C_DIS
LIN {X -13.7434,Y -92.9846,Z 93,A -103.8044,B 24.9379,C -1.8206,E1 24.9739,E2 189.1347} C_DIS
LIN {X -17.2238,Y -92.4026,Z 93,A -105.1894,B 24.936,C -1.8473,E1 24.9703,E2 190.4578} C_DIS
LIN {X -20.4886,Y -91.7333,Z 93,A -107.5801,B 24.9368,C -1.836,E1 24.9637,E2 192.8782} C_DIS
LIN {X -25.8658,Y -90.3646,Z 93,A -110.7023,B 24.9361,C -1.8468,E1 24.9553,E2 195.9794} C_DIS
LIN {X -28.7016,Y -89.5043,Z 93,A -112.918,B 24.9369,C -1.8344,E1 24.9493,E2 198.2284} C_DIS
LIN {X -34.7163,Y -87.3479,Z 93,A -116.4102,B 24.9358,C -1.8514,E1 24.9403,E2 201.6876} C_DIS
LIN {X -37.6801,Y -86.1102,Z 93,A -118.5064,B 24.9359,C -1.8488,E1 24.9348,E2 203.7946} C_DIS
LIN {X -42.2344,Y -83.9719,Z 93,A -121.5557,B 24.9356,C -1.853,E1 24.9272,E2 206.8419} C_DIS
LIN {X -49.0898,Y -80.1563,Z 93,A -126.3015,B 24.9351,C -1.8608,E1 24.9157,E2 211.583} C_DIS
LIN {X -52.11,Y -78.2271,Z 93,A -128.5985,B 24.9351,C -1.8605,E1 24.9102,E2 213.888} C_DIS
LIN {X -54.9787,Y -76.2384,Z 93,A -130.5685,B 24.9345,C -1.8692,E1 24.9058,E2 215.8441} C_DIS
LIN {X -57.9172,Y -74.0292,Z 93,A -134.0622,B 24.937,C -1.8331,E1 24.8979,E2 219.4367} C_DIS
LIN {X -62.1993,Y -70.4715,Z 93,A -136.3845,B 24.9342,C -1.8737,E1 24.8931,E2 221.6713} C_DIS
LIN {X -64.5353,Y -68.3372,Z 93,A -138.1894,B 24.9336,C -1.8816,E1 24.8895,E2 223.4648} C_DIS
LIN {X -66.8516,Y -66.0727,Z 93,A -140.2709,B 24.9336,C -1.8823,E1 24.8853,E2 225.5534} C_DIS
LIN {X -70.0614,Y -62.6589,Z 93,A -142.9354,B 24.9327,C -1.8947,E1 24.8803,E2 228.2} C_DIS
LIN {X -71.6869,Y -60.7929,Z 93,A -144.7516,B 24.9332,C -1.8884,E1 24.8769,E2 230.0396} C_DIS
LIN {X -73.8643,Y -58.1277,Z 93,A -146.858,B 24.9328,C -1.893,E1 24.8733,E2 232.1447} C_DIS
LIN {X -76.0276,Y -55.2688,Z 93,A -148.9615,B 24.9323,C -1.901,E1 24.8698,E2 234.2394} C_DIS
LIN {X -77.8416,Y -52.6823,Z 93,A -151.0356,B 24.9323,C -1.9012,E1 24.8665,E2 236.3234} C_DIS
LIN {X -80.6357,Y -48.3003,Z 93,A -153.9544,B 24.9311,C -1.9172,E1 24.8622,E2 239.2188} C_DIS
LIN {X -81.9362,Y -46.0571,Z 93,A -155.6544,B 24.9311,C -1.9177,E1 24.8598,E2 240.9265} C_DIS
LIN {X -83.3157,Y -43.5125,Z 93,A -157.5177,B 24.9309,C -1.9194,E1 24.8574,E2 242.7956} C_DIS
LIN {X -85.0563,Y -40.0032,Z 93,A -159.5997,B 24.9298,C -1.9356,E1 24.8549,E2 244.8501} C_DIS
LIN {X -86.5208,Y -36.7281,Z 93,A -162.6379,B 24.9312,C -1.9154,E1 24.8514,E2 247.9532} C_DIS
LIN {X -87.865,Y -33.3838,Z 93,A -164.0505,B 24.929,C -1.9461,E1 24.8501,E2 249.3006} C_DIS
LIN {X -88.9857,Y -30.2712,Z 93,A -166.3236,B 24.9291,C -1.9441,E1 24.8479,E2 251.5915} C_DIS
LIN {X -90.0311,Y -27.0039,Z 93,A -168.434,B 24.9287,C -1.9497,E1 24.8462,E2 253.7005} C_DIS
LIN {X -90.9462,Y -23.7413,Z 93,A -170.4859,B 24.9282,C -1.9564,E1 24.8447,E2 255.7484} C_DIS
LIN {X -91.6622,Y -20.8065,Z 93,A -172.4305,B 24.9281,C -1.9589,E1 24.8434,E2 257.6984} C_DIS
LIN {X -92.3966,Y -17.259,Z 93,A -174.6676,B 24.9276,C -1.9649,E1 24.8422,E2 259.9346} C_DIS
LIN {X -92.9853,Y -13.7387,Z 93,A -176.8702,B 24.9272,C -1.9709,E1 24.8413,E2 262.1359} C_DIS
LIN {X -93.6226,Y -8.3443,Z 93,A -179.9455,B 24.9259,C -1.9886,E1 24.8404,E2 265.1874} C_DIS
LIN {X -93.9372,Y -3.2433,Z 93,A 176.7405,B 24.9256,C -1.9924,E1 24.8399,E2 268.5122} C_DIS
LIN {X -93.9944,Y -0.2836,Z 93,A 174.773,B 24.9256,C -1.9932,E1 24.8398,E2 270.4897} C_DIS
LIN {X -93.913,Y 3.8858,Z 93,A 171.6702,B 24.9262,C -1.9843,E1 24.8401,E2 273.6323} C_DIS
LIN {X -93.647,Y 8.08,Z 93,A 169.9562,B 24.9236,C -2.0183,E1 24.8405,E2 275.2755} C_DIS
LIN {X -92.8896,Y 14.3614,Z 93,A 166.0625,B 24.9228,C -2.0296,E1 24.8418,E2 279.1657} C_DIS
LIN {X -91.7686,Y 20.3312,Z 93,A 162.307,B 24.922,C -2.0397,E1 24.8438,E2 282.9192} C_DIS
LIN {X -90.9832,Y 23.597,Z 93,A 159.9526,B 24.9222,C -2.0368,E1 24.8454,E2 285.2943} C_DIS
LIN {X -89.8253,Y 27.6799,Z 93,A 157.1768,B 24.922,C -2.0391,E1 24.8476,E2 288.0806} C_DIS
LIN {X -88.3251,Y 32.1467,Z 93,A 154.6592,B 24.9205,C -2.0588,E1 24.8499,E2 290.5653} C_DIS
LIN {X -87.014,Y 35.543,Z 93,A 152.0494,B 24.9209,C -2.0537,E1 24.8527,E2 293.2022} C_DIS
LIN {X -85.5979,Y 38.8302,Z 93,A 150.0953,B 24.9199,C -2.0672,E1 24.8549,E2 295.1347} C_DIS
LIN {X -83.2798,Y 43.5806,Z 93,A 146.8839,B 24.9191,C -2.077,E1 24.8589,E2 298.3399} C_DIS
LIN {X -80.9207,Y 47.8182,Z 93,A 144.1592,B 24.9179,C -2.0927,E1 24.8626,E2 301.0414} C_DIS
LIN {X -79.6021,Y 49.9829,Z 93,A 142.517,B 24.9178,C -2.0941,E1 24.865,E2 302.6887} C_DIS
LIN {X -77.821,Y 52.7127,Z 93,A 139.9919,B 24.9186,C -2.083,E1 24.869,E2 305.2529} C_DIS
LIN {X -75.3436,Y 56.1977,Z 93,A 137.7721,B 24.9171,C -2.102,E1 24.8726,E2 307.4383} C_DIS
LIN {X -73.1039,Y 59.081,Z 93,A 135.5738,B 24.9166,C -2.1087,E1 24.8764,E2 309.6308} C_DIS
LIN {X -70.8742,Y 61.7382,Z 93,A 133.4271,B 24.9163,C -2.1131,E1 24.8803,E2 311.7768} C_DIS
LIN {X -68.4311,Y 64.4355,Z 93,A 131.2383,B 24.9157,C -2.1196,E1 24.8844,E2 313.9598} C_DIS
LIN {X -65.7987,Y 67.1222,Z 93,A 128.8889,B 24.9154,C -2.1233,E1 24.889,E2 316.3102} C_DIS
LIN {X -63.3368,Y 69.4497,Z 93,A 126.7989,B 24.9151,C -2.1273,E1 24.8933,E2 318.3992} C_DIS
LIN {X -60.7372,Y 71.7343,Z 93,A 124.5016,B 24.9152,C -2.1262,E1 24.8982,E2 320.7082} C_DIS
LIN {X -57.9534,Y 74.0021,Z 93,A 122.6365,B 24.914,C -2.1411,E1 24.9022,E2 322.5447} C_DIS
LIN {X -55.4047,Y 75.9281,Z 93,A 120.6304,B 24.9138,C -2.1433,E1 24.9067,E2 324.5528} C_DIS
LIN {X -51.4618,Y 78.6545,Z 93,A 117.6384,B 24.9136,C -2.1468,E1 24.9136,E2 327.5465} C_DIS
LIN {X -48.8138,Y 80.324,Z 93,A 115.658,B 24.9135,C -2.148,E1 24.9183,E2 329.5301} C_DIS
LIN {X -45.474,Y 82.2619,Z 93,A 113.3409,B 24.913,C -2.1533,E1 24.9239,E2 331.8414} C_DIS
LIN {X -42.3472,Y 83.9147,Z 93,A 110.5205,B 24.9145,C -2.1356,E1 24.931,E2 334.7116} C_DIS
LIN {X -38.8405,Y 85.5933,Z 93,A 108.9603,B 24.9121,C -2.1652,E1 24.9348,E2 336.2053} C_DIS
LIN {X -36.3489,Y 86.6806,Z 93,A 106.8124,B 24.9132,C -2.1517,E1 24.9404,E2 338.3901} C_DIS
LIN {X -32.458,Y 88.2115,Z 93,A 104.1286,B 24.9132,C -2.1507,E1 24.9475,E2 341.0819} C_DIS
LIN {X -29.3811,Y 89.2844,Z 93,A 102.5142,B 24.9121,C -2.1651,E1 24.9517,E2 342.6651} C_DIS
LIN {X -25.9448,Y 90.3422,Z 93,A 99.338,B 24.9145,C -2.1356,E1 24.9604,E2 345.9165} C_DIS
LIN {X -20.7682,Y 91.671,Z 93,A 97.3177,B 24.9109,C -2.179,E1 24.9656,E2 347.8366} C_DIS
LIN {X -17.3626,Y 92.3762,Z 93,A 94.4066,B 24.9129,C -2.1547,E1 24.9738,E2 350.8086} C_DIS
LIN {X -13.6632,Y 92.996,Z 93,A 92.9161,B 24.9107,C -2.1825,E1 24.9777,E2 352.2344} C_DIS
LIN {X -7.7397,Y 93.6744,Z 93,A 89.3871,B 24.9102,C -2.1879,E1 24.9875,E2 355.7526} C_DIS
LIN {X -2.6789,Y 93.9553,Z 93,A 85.9242,B 24.9111,C -2.1765,E1 24.9972,E2 359.2436} C_DIS
LIN {X 2.2573,Y 93.9677,Z 93,A 83.1791,B 24.9104,C -2.1859,E1 25.0048,E2 361.9662} C_DIS
LIN {X 5.859,Y 93.8117,Z 93,A 80.33,B 24.9122,C -2.164,E1 25.0129,E2 364.8662} C_DIS
LIN {X 9.9122,Y 93.4693,Z 93,A 78.1305,B 24.9114,C -2.1732,E1 25.0189,E2 367.0426} C_DIS
LIN {X 14.6295,Y 92.8482,Z 93,A 75.2562,B 24.9114,C -2.1732,E1 25.0269,E2 369.914} C_DIS
LIN {X 20.2982,Y 91.7758,Z 93,A 71.6729,B 24.9117,C -2.1695,E1 25.0367,E2 373.5021} C_DIS
LIN {X 23.5798,Y 90.9877,Z 93,A 69.7583,B 24.9114,C -2.1732,E1 25.0418,E2 375.405} C_DIS
LIN {X 27.1054,Y 90.001,Z 93,A 67.5357,B 24.9115,C -2.1719,E1 25.0478,E2 377.6268} C_DIS
LIN {X 30.5268,Y 88.8995,Z 93,A 65.4334,B 24.9115,C -2.1732,E1 25.0534,E2 379.7221} C_DIS
LIN {X 32.5794,Y 88.1673,Z 93,A 63.9511,B 24.912,C -2.1666,E1 25.0573,E2 381.2169} C_DIS
LIN {X 36.2033,Y 86.7419,Z 93,A 61.1144,B 24.9135,C -2.1481,E1 25.0647,E2 384.091} C_DIS
LIN {X 39.6104,Y 85.2394,Z 93,A 59.8486,B 24.9108,C -2.1806,E1 25.0677,E2 385.2766} C_DIS
LIN {X 43.5729,Y 83.2839,Z 93,A 56.3653,B 24.9134,C -2.1494,E1 25.0766,E2 388.8243} C_DIS
LIN {X 47.2638,Y 81.2473,Z 93,A 54.0623,B 24.9129,C -2.1551,E1 25.0821,E2 391.107} C_DIS
LIN {X 50.5021,Y 79.2741,Z 93,A 51.3843,B 24.9142,C -2.1386,E1 25.0885,E2 393.8153} C_DIS
LIN {X 53.3761,Y 77.3682,Z 93,A 50.0711,B 24.9122,C -2.1632,E1 25.0914,E2 395.0659} C_DIS
LIN {X 55.5202,Y 75.8435,Z 93,A 47.0739,B 24.9164,C -2.111,E1 25.0984,E2 398.176} C_DIS
LIN {X 59.9744,Y 72.3728,Z 93,A 45.1593,B 24.9126,C -2.159,E1 25.1023,E2 399.9698} C_DIS
LIN {X 61.8293,Y 70.7946,Z 93,A 43.3298,B 24.9138,C -2.1437,E1 25.1062,E2 401.8284} C_DIS
LIN {X 64.5206,Y 68.351,Z 93,A 41.2736,B 24.9138,C -2.1449,E1 25.1104,E2 403.8733} C_DIS
LIN {X 66.4611,Y 66.468,Z 93,A 39.2175,B 24.9152,C -2.1267,E1 25.1146,E2 405.9639} C_DIS
LIN {X 71.1557,Y 61.4158,Z 93,A 35.4173,B 24.9148,C -2.1319,E1 25.1217,E2 409.7349} C_DIS
LIN {X 73.6334,Y 58.4199,Z 93,A 32.1395,B 24.9178,C -2.0934,E1 25.1276,E2 413.0885} C_DIS
LIN {X 76.283,Y 54.9163,Z 93,A 28.9615,B 24.9197,C -2.0687,E1 25.1328,E2 416.3093} C_DIS
LIN {X 79.7211,Y 49.7924,Z 93,A 26.5771,B 24.9166,C -2.109,E1 25.1362,E2 418.5865} C_DIS
LIN {X 81.4201,Y 46.9631,Z 93,A 23.7684,B 24.9193,C -2.0745,E1 25.1402,E2 421.4624} C_DIS
LIN {X 83.4807,Y 43.1965,Z 93,A 22.0918,B 24.9172,C -2.1018,E1 25.1423,E2 423.0656} C_DIS
LIN {X 85.1978,Y 39.6997,Z 93,A 19.5678,B 24.9181,C -2.0897,E1 25.1454,E2 425.6047} C_DIS
LIN {X 87.2206,Y 35.0356,Z 93,A 16.5848,B 24.9185,C -2.085,E1 25.1487,E2 428.5822} C_DIS
LIN {X 88.3155,Y 32.1731,Z 93,A 14.5868,B 24.9193,C -2.0747,E1 25.1506,E2 430.5934} C_DIS
LIN {X 90.2431,Y 26.2869,Z 93,A 10.8576,B 24.92,C -2.0651,E1 25.1538,E2 434.3241} C_DIS
LIN {X 91.4927,Y 21.5372,Z 93,A 7.7862,B 24.921,C -2.0531,E1 25.1559,E2 437.4062} C_DIS
LIN {X 92.7049,Y 15.5091,Z 93,A 4.3635,B 24.921,C -2.0536,E1 25.1577,E2 440.8076} C_DIS
LIN {X 93.1021,Y 12.9161,Z 93,A 1.9041,B 24.9238,C -2.0165,E1 25.1587,E2 443.3402} C_DIS
LIN {X 93.5671,Y 8.9463,Z 93,A 0.4073,B 24.9217,C -2.0438,E1 25.1591,E2 444.7636} C_DIS
LIN {X 93.8438,Y 5.2996,Z 93,A -2.0233,B 24.9228,C -2.0291,E1 25.1596,E2 447.2144} C_DIS
LIN {X 93.9744,Y 1.889,Z 93,A -4.1176,B 24.9233,C -2.022,E1 25.1598,E2 449.3132} C_DIS
LIN {X 93.9747,Y -1.8759,Z 93,A -6.6381,B 24.9245,C -2.0061,E1 25.1597,E2 451.8561} C_DIS
LIN {X 93.8242,Y -5.6539,Z 93,A -8.5887,B 24.9241,C -2.012,E1 25.1594,E2 453.7813} C_DIS
LIN {X 93.584,Y -8.7634,Z 93,A -10.5316,B 24.9247,C -2.0043,E1 25.159,E2 455.7308} C_DIS
LIN {X 93.0078,Y -13.5801,Z 93,A -13.399,B 24.9251,C -1.9982,E1 25.158,E2 458.5957} C_DIS
LIN {X 92.1955,Y -18.3022,Z 93,A -16.1969,B 24.9255,C -1.9934,E1 25.1566,E2 461.3885} C_DIS
LIN {X 91.3709,Y -22.0488,Z 93,A -18.7587,B 24.9267,C -1.9776,E1 25.155,E2 463.9727} C_DIS
LIN {X 90.4707,Y -25.4913,Z 93,A -21.467,B 24.9287,C -1.9506,E1 25.153,E2 466.7291} C_DIS
LIN {X 89.4152,Y -28.9769,Z 93,A -23.0543,B 24.9274,C -1.9673,E1 25.1517,E2 468.2681} C_DIS
LIN {X 87.7141,Y -33.7825,Z 93,A -26.0705,B 24.9279,C -1.9611,E1 25.1488,E2 471.282} C_DIS
LIN {X 86.2915,Y -37.2643,Z 93,A -28.5403,B 24.9289,C -1.9474,E1 25.1461,E2 473.7704} C_DIS
LIN {X 84.8165,Y -40.5087,Z 93,A -30.6507,B 24.9292,C -1.9432,E1 25.1436,E2 475.8793} C_DIS
LIN {X 83.2522,Y -43.633,Z 93,A -33.1641,B 24.9307,C -1.9227,E1 25.1404,E2 478.428} C_DIS
LIN {X 81.3183,Y -47.1402,Z 93,A -35.2463,B 24.9302,C -1.9289,E1 25.1375,E2 480.4846} C_DIS
LIN {X 79.5765,Y -50.0239,Z 93,A -38.1321,B 24.9329,C -1.8923,E1 25.1332,E2 483.4423} C_DIS
LIN {X 76.8366,Y -54.1398,Z 93,A -40.2799,B 24.9312,C -1.9159,E1 25.1298,E2 485.5238} C_DIS
LIN {X 73.7554,Y -58.2656,Z 93,A -43.4806,B 24.932,C -1.9052,E1 25.1244,E2 488.7346} C_DIS
LIN {X 69.6205,Y -63.1507,Z 93,A -47.0555,B 24.9318,C -1.9072,E1 25.1179,E2 492.2886} C_DIS
LIN {X 67.746,Y -65.1554,Z 93,A -49.5285,B 24.9342,C -1.8736,E1 25.113,E2 494.8301} C_DIS
Enddeposition()
END
